# B&R Automation Studio project Parker_BMM_ST_V5_3147_V12 (part 31)

#### modem.c
```c
/********************************************************************
 * COPYRIGHT --  B&R China
 ********************************************************************
 * Program: modem
 * File: modem.c
 * Author: lijianjun
 * Created: March 06, 2013
 ********************************************************************
 * Implementation of program modem --- modem remote communication  control
 ********************************************************************/

#ifdef _DEFAULT_INCLUDES
	#include <AsDefault.h>
#endif

#include <bur/plctypes.h>
#include <string.h>
#include "edge.h"

/**************************************************************************************
** 					 	     define 								                 **
**************************************************************************************/
#define	BRTRSM_COMMAND_CHAR_MAXCOUT			20
#define	BRTRSM_COMMAND_MAXCOUT					20

#define  BRTRSM_EXCHANGEDATA_CHAR_MAXCOUT		64

#define  BRTRSM_ERR_FUB_BUSY		0xFFFF

/**************************************************************************************
** 					 	     function 								                 **
**************************************************************************************/
UINT	BRFindString(char * p,char * str);

/**************************************************************************************
**     	        		I N I T U P  O F   T H E   T A S K 		 				     **
**************************************************************************************/
 _INIT void init ( void )
 {
	 BRInitStep		= 1000;
	 BRStep			= 0;
 }

 /**************************************************************************************
**        				C Y C L I C   P A R T   O F   T H E   T A S K  				 **
**************************************************************************************/

 _CYCLIC void cyclic ( void )
 {

	switch	(BRInitStep)
	{
		case 1000:

			cmdModem		=0;

			strcpy(FmDevice,"IF1");
			#ifdef __i386__

			strcpy(FmMode,"/PHY=RS232 /BD=57600 /PA=N /DB=8 /SB=1");

			#else

			strcpy(FmMode,"57600,N,8,1,RS232");

			#endif

			i	=0;

			strcpy(AcT[i++].Command,"AT&F");	  /* DEFAULT SETTING  */
			strcpy(AcT[i++].Command,"ATS0=1");
			strcpy(AcT[i++].Command,"ATS37=9");
			strcpy(AcT[i++].Command,"AT&C0");
			strcpy(AcT[i++].Command,"AT&D0");
			strcpy(AcT[i++].Command,"AT&K0");
			strcpy(AcT[i++].Command,"AT&Q0");
			strcpy(AcT[i++].Command,"AT&W0");
			strcpy(AcT[i++].Command,"AT&Y0");

			ATCommandCount = i;

			BRInitStep	   = 2000;

			break;
		case 2000:
			if (0 == BRStep && 1 == cmdModem)
			{
				gMachineInfo.Modem_Ok	= 0;
				BRStep		= 1000;
				BRInitStep	= 3000;
			}
			break;
		case 3000:
			Status	=BRFindString(BRReadBuf,BRWriteBuf);
			break;
		default:
         break;
	}
	switch	(BRStep)
	{
		case 1000:

			BRFRMxopen.device	= (unsigned long)&FmDevice;
			BRFRMxopen.mode		= (unsigned long)&FmMode;
			BRFRMxopen.enable	= 1;

			FRM_xopen(&BRFRMxopen);

			if(0 == BRFRMxopen.status)
			{
				BRStep	= 2000;
			}

			break;

		case 2000:

			BRFRMctrl.enable	= 1;
			BRFRMctrl.ident		= BRFRMxopen.ident;
			BRFRMctrl.ioctrl	= 0x12;
			BRFRMctrl.inarg		= 1;

			FRM_ctrl(&BRFRMctrl);

			BRFRMctrl.enable	= 1;
			BRFRMctrl.ident		= BRFRMxopen.ident;
			BRFRMctrl.ioctrl	= 0x27;

			FRM_ctrl(&BRFRMctrl);

			BRStep	= 3000;

			break;
		case 3000:

			memset(BRWriteBuf,0,BRTRSM_EXCHANGEDATA_CHAR_MAXCOUT);
			strcpy(BRWriteBuf,"AT&F");
			BRWriteBuf[4]	= 0x0D;
			BRWriteBuf[5]	= 0x00;

			BRFRMwrite.enable	= 1;
			BRFRMwrite.ident	= BRFRMxopen.ident;
			BRFRMwrite.buffer	= (unsigned long)BRWriteBuf;
			BRFRMwrite.buflng	= strlen(BRWriteBuf);

			FRM_write(&BRFRMwrite);

			if(0 == BRFRMwrite.status)
			{
				BRStep = 3200;
			}

			break;
		case 3200:
			memset(BRWriteBuf,0,BRTRSM_EXCHANGEDATA_CHAR_MAXCOUT);
			strcpy(BRWriteBuf,"ATE0");
			BRWriteBuf[4]	= 0x0D;
			BRWriteBuf[5]	= 0x00;

			BRFRMwrite.enable	= 1;
			BRFRMwrite.ident	= BRFRMxopen.ident;
			BRFRMwrite.buffer	= (unsigned long)BRWriteBuf;
			BRFRMwrite.buflng	= strlen(BRWriteBuf);

			FRM_write(&BRFRMwrite);

			if(0 == BRFRMwrite.status)
			{
				BRStep = 3600;
			}

			break;
		case 3600:
			memset(BRWriteBuf,0,BRTRSM_EXCHANGEDATA_CHAR_MAXCOUT);
			strcpy(BRWriteBuf,"AT&Q0");
			BRWriteBuf[4]	= 0x0D;
			BRWriteBuf[5]	= 0x00;

			BRFRMwrite.enable	= 1;
			BRFRMwrite.ident	= BRFRMxopen.ident;
			BRFRMwrite.buffer	= (unsigned long)BRWriteBuf;
			BRFRMwrite.buflng	= strlen(BRWriteBuf);

			FRM_write(&BRFRMwrite);

			if(0 == BRFRMwrite.status)
			{
				BRStep = 4000;
			}
			break;
		case 4000:

			BRFRMread.enable = 1;
			BRFRMread.ident	 = BRFRMxopen.ident;

			FRM_read(&BRFRMread);

			if(0 == BRFRMread.status)
			{
				if(BRFRMread.buflng<=BRTRSM_EXCHANGEDATA_CHAR_MAXCOUT)
				{
					memcpy(BRReadBuf,(void*)BRFRMread.buffer,BRFRMread.buflng);		/* copy received data */

					BRFRMrbuf.enable	= 1;
					BRFRMrbuf.ident		= BRFRMxopen.ident;
					BRFRMrbuf.buffer	= BRFRMread.buffer;
					BRFRMrbuf.buflng	= BRFRMread.buflng;

					FRM_rbuf(&BRFRMrbuf);											/* release buffer again */

					if(BRFindString(BRReadBuf,"OK")==1)
					{
						CurrentAT	= 0;
						BRStep		= 5000;
					}
					else
					{
						BRStep		= 3000;
					}
				}
			}

			break;
		case 5000:

			memset(BRWriteBuf,0,BRTRSM_EXCHANGEDATA_CHAR_MAXCOUT);
			strcpy(BRWriteBuf,AcT[CurrentAT].Command);
			TempLength	=strlen(BRWriteBuf);
			BRWriteBuf[TempLength]		= 0x0D;
			BRWriteBuf[TempLength+1]	= 0x00;

			TempLength++;

			BRFRMwrite.enable		=1;
			BRFRMwrite.ident		=BRFRMxopen.ident;
			BRFRMwrite.buffer		=(unsigned long)BRWriteBuf;
			BRFRMwrite.buflng		=strlen(BRWriteBuf);

			FRM_write(&BRFRMwrite);

			if(BRFRMwrite.status==0)
			{
				BRStep			=6000;
			}

			break;
		case 6000:

			BRFRMread.enable		=1;
			BRFRMread.ident			=BRFRMxopen.ident;

			FRM_read(&BRFRMread);

			if(BRFRMread.status==0)
			{
				if(BRFRMread.buflng<=BRTRSM_EXCHANGEDATA_CHAR_MAXCOUT)
				{
					memcpy(BRReadBuf,(void*)BRFRMread.buffer,BRFRMread.buflng);		/* copy received data */

					BRFRMrbuf.enable	=1;
					BRFRMrbuf.ident		=BRFRMxopen.ident;
					BRFRMrbuf.buffer	=BRFRMread.buffer;
					BRFRMrbuf.buflng	=BRFRMread.buflng;

					FRM_rbuf(&BRFRMrbuf);											/* release buffer again */

					if(BRFindString(BRReadBuf,"OK")==1)
					{
						CurrentAT++;
						if(CurrentAT>=ATCommandCount)
						{
							BRStep		=7000;
							break;
						}
					}
					BRStep			=5000;

				}
			}
			break;
		case 7000:

			BRFRMclose.enable	=1;
			BRFRMclose.ident	=BRFRMxopen.ident;

			FRM_close(&BRFRMclose);

			BRStep	= 8000;

			break;

		case 8000:
			cmdModem		=0;
			gMachineInfo.Modem_Ok =1;
			BRStep		    =0;

			break;
		default:
         break;
	}

 }
/**************************************************************************************
** 					 	     function 								                 **
**************************************************************************************/
UINT	BRFindString(char * p,char * str)
{
   UINT pLength,strLength,i,j;

   pLength	   =strlen(p);
   strLength	=strlen(str);

   if(strLength==0)
      return 0;
   if(pLength==0)
      return 0;

   j		=0;

   for(i=0;i<pLength;i++)
   {
      if(p[i]==str[j])
      {
         j++;
         if(j>=strLength)
         {
            return 1;
         }
      }
      else
      {
         j		=0;
         if(p[i]==str[j])
         {
            j++;
            if(j>=strLength)
            {
               return 1;
            }
         }
      }
   }

   return 0;
}
```

#### modem.var
```iecst
VAR
	cmdModem : BOOL;
	BRInitStep : UINT;
	BRStep : UINT;
	Status : UINT;
	i : UINT;
	ATCommandCount : UINT;
	CurrentAT : UINT;
	TempLength : UINT;
	BRReadBuf : STRING[80];
	BRWriteBuf : STRING[80];
	FmDevice : STRING[80];
	FmMode : STRING[80];
	BRFRMwrite : FRM_write;
	BRFRMread : FRM_read;
	BRFRMctrl : FRM_ctrl;
	BRFRMxopen : FRM_xopen;
	BRFRMrbuf : FRM_rbuf;
	BRFRMclose : FRM_close;
	AcT : ARRAY[0..19] OF BRTransfer;
END_VAR
```

### Program Logical/comm/mbusMaster (ANSIC, version 1.00.0) - communication with frequency inventor

#### mbusMaster.c - Implementation code
```c
/********************************************************************
 * COPYRIGHT --
 ********************************************************************
 * Program: mbusMaster
 * File: mbusMaster.c
 * Author: lij
 * Created: December 12, 2014
 ********************************************************************
 * Implementation of program mbusMaster
 ********************************************************************/

#include <bur/plctypes.h>
#include <string.h>

#ifdef _DEFAULT_INCLUDES
	#include <AsDefault.h>
#endif

#define	_AR_I386_AUTOMATION_STUDIO_   1

void _INIT mbusMasterINIT(void)
{
	/* TODO: Add code here */

   ascii = 0;    /* 0 = RTU / 1 = ASCII */

#ifdef _AR_I386_AUTOMATION_STUDIO_
   strcpy(sDeviceName, "SL1.SS1.IF1.ST2.IF1");
   if (!ascii)
   {
      strcpy(sModeName, "PHY=RS485 /BD=19200 /PA=O /DB=8");
   }
   else
   {
      strcpy(sModeName, "PHY=RS485 /BD=19200 /PA=O /DB=7");
   }
#else
   strcpy(sDeviceName, "SS1.IF1");
   if (!ascii)
   {
      strcpy(sModeName, "RS232,19200,E,8,1");
   }
   else
   {
      strcpy(sModeName, "RS232,19200,E,8,1");
   }
#endif

   strcpy(sConfigName, "mb_cmd");

   timeout  = 500; /* 500ms */

   /* modbus - Slave open */
   MOpen.enable   = 1;
   MOpen.pDevice  = (UDINT) &sDeviceName[0];
   MOpen.pMode    = (UDINT) &sModeName[0];
   MOpen.pConfig  = (UDINT) &sConfigName[0];
   MOpen.timeout  = timeout;
   MOpen.ascii = ascii;

   MBMOpen(&MOpen);

   statusMOpen = MOpen.status;
   if (!statusMOpen)
   {
      ident    = MOpen.ident;
      fMOpen   = 0;
      fMaster  = 1;
      fMClose  = 0;
   }
   else
   {
      fMaster = 0;
      ident   = 0;
      fMOpen  = 1;
   }

   fMClose = 0;
}

void _CYCLIC mbusMasterCYCLIC(void)
{
	/* TODO: Add code here */

   if(fMOpen)
   {
      /* modbus - Master open */
      MOpen.enable   = 1;
      MOpen.pDevice  = (UDINT) &sDeviceName[0];
      MOpen.pMode    = (UDINT) &sModeName[0];
      MOpen.pConfig  = (UDINT) &sConfigName[0];
      MOpen.timeout  = timeout;
      MOpen.ascii    = ascii;

      MBMOpen(&MOpen);

      statusMOpen = MOpen.status;
      if (!statusMOpen)
      {
         ident   = MOpen.ident;
         fMOpen  = 0;
         fMaster = 1;
         fMClose = 0;
      }
      else
      {
         fMaster = 0;
         ident   = 0;
         fMOpen  = 1;
      }
   }

   if(fMaster)
   {
      /* modbus - Master */
      Master.enable = 1;
      Master.ident  = ident;
      MBMaster(&Master);

      statusMaster= Master.status;
      execute     = Master.execute;
      recordnum   = Master.recordnum;

      if (!statusMaster)
      {
         fMaster = 1;
      }
   }

   if(fMClose)
   {
      fMaster = 0;
      fMClose = 0;

      /* modbus - Master close */
      MClose.enable = 1;
      MClose.ident  = ident;
      MBMClose(&MClose);

      statusMClose = MClose.status;
      if (!statusMClose)
      {
         ident  = 0;
         fMOpen = 0;
      }
   }
}

void _EXIT mbusMasterEXIT(void)
{
	/* TODO: Add code here */

   MClose.enable   = 1;
   MClose.ident    = ident;
   MBMClose(&MClose);
}
```

#### mbusMaster.var - Local variables
```iecst
(********************************************************************
 * COPYRIGHT --
 ********************************************************************
 * Program: mbusMaster
 * File: mbusMaster.var
 * Author: lij
 * Created: December 12, 2014
 ********************************************************************
 * Local variables of program mbusMaster
 ********************************************************************)
VAR
	MOpen : MBMOpen;
	Master : MBMaster;
	MClose : MBMClose;
	fMOpen : BOOL;
	fMaster : BOOL;
	fMClose : BOOL;
	ascii : USINT;
	statusMOpen : UINT;
	statusMaster : UINT;
	statusMClose : UINT;
	timeout : UINT;
	ident : UDINT;
	execute : UDINT;
	recordnum : UDINT;
	sDeviceName : STRING[80];
	sModeName : STRING[80];
	sConfigName : STRING[80];
END_VAR
```

### Data object Logical/comm/mb_cmd (Simple) - A simple data object.

#### mb_cmd.dat
```
(********************************************************************
 * COPYRIGHT --
 ********************************************************************
 * Data object: mb_cmd
 * File: mb_cmd.dat
 * Author: lij
 * Created: December 12, 2014
 ********************************************************************
 * Data object file: mb_cmd.dat
 ********************************************************************)
; ---------------------------------------------------------------------------
; SanKen VM06 系列选件板
; MODBUS-RTU
; MODBUS command table
; ---------------------------------------------------------------------------
; Modbus Function Code description
; ---------------------------------------------------------------------------
; 功能编码	名称
; 0x03	    读控制继电器
; 0x04	    读输入继电器
; 0x06	    写信号继电器
; 0x10	    Preset Multiple Register
; ---------------------------------------------------------------------------
; ---------------------------------------------------------------------------

; ---------------------------------------------------------------------------
; ---------------------------------------------------------------------------
;         1         2         3                        1         2         3
;1234567890123456789012345678901              1234567890123456789012345678901
;"                               ", 03, $02, "LocalPV3                       ", 0000, 0800    ;read from MB4[x], block read supported
;"                               ", 06, $02, "LocalPV6[0]                    ", 0000, 0001    ;function code 6:write to MB4[x]
;"                               ", 16, $02, "LocalPV16                      ", 0000, 0200    ;EventPV16
;|                                 |    |    |                                  |     |
;|                                 |    |    |                                  |     |
;Event variable                    |    |    Variable name on this station      |     Data Length to be read or written[WORD]
;                                  |    Node number [BYTE](server?)             Modbus offset
;                                  Modbus function code [BYTE]                  on slave station [WORD]
; ---------------------------------------------------------------------------
; ---------------------------------------------------------------------------

;1234567890123456789012345678901             1234567890123456789012345678901

;Slave 1:	Main   Extruder		SanKen VM06-0150-N4
"                               ", 06, $01, "gMbusCom[0].WriteFrequency      ", 1000, 0001
"                               ", 06, $01, "gMbusCom[0].WriteCommand        ", 1001, 0001
"                               ", 06, $01, "gMbusCom[0].WriteAckAlarm       ", 1002, 0001
"                               ", 03, $01, "gMbusCom[0].ReadCurrent         ", 2003, 0001
"                               ", 03, $01, "gMbusCom[0].ReadFrequency       ", 2002, 0001
"                               ", 03, $01, "gMbusCom[0].ReadVoltage         ", 2014, 0001
"                               ", 03, $01, "gMbusCom[0].ReadAlarmNum        ", 2000, 0001
"                               ", 03, $01, "gMbusCom[0].ReadStatus          ", 2008, 0002
; ---------------------------------------------------------------------------
; ---------------------------------------------------------------------------
;Slave 2:	AUX1   Extruder		SanKen VM06-0150-N4
"                               ", 06, $02, "gMbusCom[1].WriteFrequency      ", 1000, 0001
"                               ", 06, $02, "gMbusCom[1].WriteCommand        ", 1001, 0001
"                               ", 06, $02, "gMbusCom[1].WriteAckAlarm       ", 1002, 0001
"                               ", 03, $02, "gMbusCom[1].ReadCurrent         ", 2003, 0001
"                               ", 03, $02, "gMbusCom[1].ReadFrequency       ", 2002, 0001
"                               ", 03, $02, "gMbusCom[1].ReadVoltage         ", 2014, 0001
"                               ", 03, $02, "gMbusCom[1].ReadAlarmNum        ", 2000, 0001
"                               ", 03, $02, "gMbusCom[1].ReadStatus          ", 2008, 0002
; ---------------------------------------------------------------------------
; ---------------------------------------------------------------------------
```

### Program Logical/comm/epl (ANSIC)

#### epl.c - Init, cyclic, exit code
```c
#include <bur/plctypes.h>

#ifdef _DEFAULT_INCLUDES
	#include <AsDefault.h>
#endif

void _INIT eplInit(void)
{
	EPLInverter[0].cmd.readNode = 1;
	EPLInverter[1].cmd.readNode = 1;
	EPLInverter[2].cmd.readNode = 1;
	EPLInverter[3].cmd.readNode = 1;

	strcpy(&sDevice[0],"SL1.IF1");
	strcpy(&sDevice[1],"SL1.IF1");
	strcpy(&sDevice[2],"SL1.IF1");
	strcpy(&sDevice[3],"SL1.IF1");

	strcpy(&sDeviceAExtr,"SL1.IF1");

	uIndexOffset = 7;

	/*Albert*/

	uCountTimerA = 100;/*1 second*/
	uCountTimerB = 100;/*1 second*/
	uCountTimerC = 100;/*1 second*/
	uCountTimerV = 100;/*1 second*/

	uIndexA = 0;
	uIndexB = 0;
	uIndexC = 0;
	uIndexV = 0;
}

void _CYCLIC eplCyclic(void)
{
//	int i;
//	for(i=0;i<4;i++)/*For extruder A , B , C and V*/
//	{
//		if(EPLInverter[i].para.nodeNr != 0)
//		{
//			if(EPLInverter[i].state = EPL_WAIT)
//			{
//				EPLInverter[i].cmd.bReadObj = 1;/*read command*/
//				if (0 == uIndexRead[i])
//				{
//					EPLInverter[i].para.MotorPower = (INT) EPLInverter[i].para.readData;
//					uIndexRead[i] = uIndexRead[i]+10;
//					EPLInverter[i].cmd.index = 0x2002;
//					EPLInverter[i].cmd.subindex = 0x9;
//				}
//				else if (10 == EPLInverter[i].cmd.index)
//				{
//					EPLInverter[i].para.MotorVoltage = (INT) EPLInverter[i].para.readData;
//					uIndexRead[i] = 0;
//					EPLInverter[i].cmd.index = 0x2002;
//					EPLInverter[i].cmd.subindex = 0xC;
//				}
//			}
//		}
//		switch (EPLInverter[i].state)
//		{
//			case EPL_WAIT: /*state to wait for user Commands*/
//
//				if(1 == EPLInverter[i].cmd.readNode)
//				{
//					EPLInverter[i].cmd.readNode = 0;
//					EPLInverter[i].state = EPL_READ_NODE;
//				}
//				else if(1 == EPLInverter[i].cmd.bReadObj)
//				{
//					EPLInverter[i].cmd.readThresholdCnt = 0;
//					EPLInverter[i].state = EPL_READ_OE;
//				}
//				else if(1 == EPLInverter[i].cmd.bWriteObj)
//				{
//					EPLInverter[i].cmd.bWriteObj = 0;
//					EPLInverter[i].state = EPL_WRITE_OE;
//				}
//
//				break;
//			case EPL_READ_NODE:/*state to read the local Powerlink node number*/
//				EPLInverter[i].fub.fnEplGetLocalNodeID.enable = 1;
//				EPLInverter[i].fub.fnEplGetLocalNodeID.pDevice = (UDINT) &sDevice[i];
//
//				if(EPLInverter[i].fub.fnEplGetLocalNodeID.status == 0)
//				{
//					EPLInverter[i].para.nodeNr = EPLInverter[i].fub.fnEplGetLocalNodeID.nodeid;
//					EPLInverter[i].fub.fnEplGetLocalNodeID.enable = 0;
//					EPLInverter[i].state = EPL_WAIT;
//				}
//				else if(EPLInverter[i].fub.fnEplGetLocalNodeID.status == ERR_FUB_BUSY)
//				{
//					EPLInverter[i].state = EPL_READ_NODE;/*creating not finished --> do again*/
//				}
//				else if (EPLInverter[i].fub.fnEplGetLocalNodeID.status == ERR_FUB_ENABLE_FALSE)
//				{
//					/*FUB is disabled*/
//				}
//				else
//				{
//					EPLInverter[i].state = EPL_ERROR;
//				}
//
//
//				break;
//			case EPL_READ_OE:/*state to read an object entry*/
//
//				EPLInverter[i].fub.fnEplSDORead.enable = 1;
//				EPLInverter[i].fub.fnEplSDORead.pDevice = (UDINT) &sDevice[i];
//				EPLInverter[i].fub.fnEplSDORead.node = uIndexOffset + i;
//				EPLInverter[i].fub.fnEplSDORead.index = EPLInverter[i].cmd.index;
//				EPLInverter[i].fub.fnEplSDORead.subindex = EPLInverter[i].cmd.subindex;
//				EPLInverter[i].fub.fnEplSDORead.pData = (UDINT) &EPLInverter[i].para.readData;
//				EPLInverter[i].fub.fnEplSDORead.datalen = sizeof(EPLInverter[i].para.readData);
//
//				if(EPLInverter[i].fub.fnEplSDORead.status == 0)
//				{
//					EPLInverter[i].fub.fnEplSDORead.enable = 0;
//					EPLInverter[i].state = EPL_WAIT;
//				}
//				else if(EPLInverter[i].fub.fnEplSDORead.status == ERR_FUB_BUSY)
//				{
//					EPLInverter[i].state = EPL_READ_OE;
//				}
//				else if(EPLInverter[i].fub.fnEplSDORead.status == ERR_FUB_ENABLE_FALSE)
//				{
//				}
//				else
//				{
//					EPLInverter[i].state = EPL_ERROR;
//				}
//
//				break;
//			case EPL_WRITE_OE:/*state to write an object entry*/
//				break;
//			case EPL_ERROR:/*State when an error occured*/
//				break;
//		}
//	}

//	if(bTestRead)
//	{
		for(i=0;i<4;i++)
		{
			if(EPLInverter[i].para.nodeNr != 0)
			{
				if(EPLInverter[i].state == EPL_WAIT)
				{
					EPLInverter[i].cmd.bReadObj = 1;/*read command*/
					if (0 == uIndexRead[i])
					{
						EPLInverter[i].para.EnergyCons = (INT) EPLInverter[i].para.readData;
//						EPLInverter[i].para.MotorPower = (INT) EPLInverter[i].para.readData;
						uIndexRead[i] = uIndexRead[i]+10;
						EPLInverter[i].cmd.index = 0x2002;
						EPLInverter[i].cmd.subindex = 0x9;
					}
					else if (10 == uIndexRead[i])
					{
						EPLInverter[i].para.MotorVoltage = (INT) EPLInverter[i].para.readData;
//						EPLInverter[i].para.MotorVoltage = (INT) EPLInverter[i].para.readData;
						uIndexRead[i] = uIndexRead[i]+10;
						EPLInverter[i].cmd.index = 0x2002;
						EPLInverter[i].cmd.subindex = 0xC;
					}
					else if(20 == uIndexRead[i])
					{
						EPLInverter[i].para.MotorPower = (INT) EPLInverter[i].para.readData;
//						EPLInverter[i].para.EnergyCons = (INT) EPLInverter[i].para.readData;
						uIndexRead[i] = 0;
						EPLInverter[i].cmd.index = 0x2002;
						EPLInverter[i].cmd.subindex = 0x1F;
					}
				}
			}
			switch (EPLInverter[i].state)
			{
				case EPL_WAIT: /*state to wait for user Commands*/

					if(1 == EPLInverter[i].cmd.readNode)
					{
						EPLInverter[i].cmd.readNode = 0;
						EPLInverter[i].state = EPL_READ_NODE;
					}
					else if(1 == EPLInverter[i].cmd.bReadObj)
					{
						EPLInverter[i].cmd.bReadObj = 0;
						EPLInverter[i].state = EPL_READ_OE;
					}
					else if(1 == EPLInverter[i].cmd.bWriteObj)
					{
						EPLInverter[i].cmd.bWriteObj = 0;
						EPLInverter[i].state = EPL_WRITE_OE;
					}

					break;
				case EPL_READ_NODE:/*state to read the local Powerlink node number*/
					EPLInverter[i].fub.fnEplGetLocalNodeID.enable = 1;
					EPLInverter[i].fub.fnEplGetLocalNodeID.pDevice = (UDINT) &sDevice[i];

					if(EPLInverter[i].fub.fnEplGetLocalNodeID.status == 0)
					{
						EPLInverter[i].para.nodeNr = EPLInverter[i].fub.fnEplGetLocalNodeID.nodeid;
						EPLInverter[i].fub.fnEplGetLocalNodeID.enable = 0;
						EPLInverter[i].state = EPL_WAIT;

					}
					else if(EPLInverter[i].fub.fnEplGetLocalNodeID.status == ERR_FUB_BUSY)
					{
						EPLInverter[i].state = EPL_READ_NODE;/*creating not finished --> do again*/
					}
					else if (EPLInverter[i].fub.fnEplGetLocalNodeID.status == ERR_FUB_ENABLE_FALSE)
					{
						/*FUB is disabled*/
					}
					else
					{
						EPLInverter[i].state = EPL_ERROR;
					}

					break;
				case EPL_READ_OE:/*state to read an object entry*/

					EPLInverter[i].fub.fnEplSDORead.enable = 1;
					EPLInverter[i].fub.fnEplSDORead.pDevice = (UDINT) &sDeviceAExtr;
					EPLInverter[i].fub.fnEplSDORead.node = uIndexOffset;
					EPLInverter[i].fub.fnEplSDORead.index = EPLInverter[i].cmd.index;
					EPLInverter[i].fub.fnEplSDORead.subindex = EPLInverter[i].cmd.subindex;
					EPLInverter[i].fub.fnEplSDORead.pData = (UDINT) &EPLInverter[i].para.readData;
					EPLInverter[i].fub.fnEplSDORead.datalen = sizeof(EPLInverter[i].para.readData);

					if(EPLInverter[i].fub.fnEplSDORead.status == 0)
					{
						EPLInverter[i].fub.fnEplSDORead.enable = 0;
						EPLInverter[i].state = EPL_WAIT;
					}
					else if(EPLInverter[i].fub.fnEplSDORead.status == ERR_FUB_BUSY)
					{
						EPLInverter[i].state = EPL_READ_OE;
					}
					else if(EPLInverter[i].fub.fnEplSDORead.status == ERR_FUB_ENABLE_FALSE)
					{
					}
					else
					{
						EPLInverter[i].state = EPL_ERROR;
					}

					break;
				case EPL_WRITE_OE:/*state to write an object entry*/
					break;
				case EPL_ERROR:/*State when an error occured*/
					break;
			}
		}
//	}
//	else
//	{
//		EPLInverter[i].fub.fnEplSDORead.enable = 0;
//		EPLInverter[i].fub.fnEplGetLocalNodeID.enable = 0;
//		EPLInverter[i].fub.fnEplSDOWrite.enable = 0;
//	}

	/*P84 Inverter power consumption*/

	/*Albert Add power consumption function*/

	/*----A Extruder-----*/
	switch (uStepPowerA)
	{
		case 0:/*Weit step*/
		if(gMachineInfo.Auto)
//			if(bTestAuto)
			{
				fnTON_10msA.IN = 1;
				fnTON_10msA.PT = uCountTimerA;
				uStepPowerA = 10;
			}
			break;
		case 10:/*Start Timer*/
			if(fnTON_10msA.Q)
			{
				fnTON_10msA.IN = 0;
				uIndexA++;
				uStepPowerA = 20;
			}
			if(0 == gMachineInfo.Auto)
//			if(0 == bTestAuto)
			{
				uIndexA	=	0;
				fnTON_10msA.IN = 0;
				uStepPowerA = 0;
			}
			break;
		case 20:/*Get value*/
			if(uIndexA > 59)
			{
				uIndexA = 0;
				rPowerTotalA += (rPowerTotalPerSecA/3600);
			}
			rPowerTotalPerSecA = 0;

			rActCurrentA[uIndexA] = gExtruderACtrl.InverterStatus.Current/10;/*Change unit from 0.1A to 1A*/
			rActVoltageA[uIndexA] = EPLInverter[0].para.MotorVoltage;
	//		rActCurrentA[uIndexA] = mcParID_Value.readPar.actCurrent;
	//		rActVoltageA[uIndexA] = mcParID_Value.readPar.actUDC;
	//		rActCurrentA[uIndexA] = rTestCurrent;
	//		rActVoltageA[uIndexA] = rTestVoltage;

			uStepPowerA = 30;

			break;
		case 30:/*Calculate*/
			rPowerA[uIndexA] = (rActCurrentA[uIndexA] * rActVoltageA[uIndexA])/1000;
			for(i_A=0;i_A<60;i_A++)
			{
				rPowerTotalPerSecA += rPowerA[i_A];
			}
			rPowerPerMinA= rPowerTotalPerSecA/60;
			uStepPowerA = 0;
			break;
	}

	/*Function call*/
	TON_10ms(&fnTON_10msA);

	/*Reset Function*/
	if(bCleanPowerA)
	{
		iClickTimeA--;
		if(iClickTimeA <= 0)
		{
			bCleanPowerA = 0;
			rPowerTotalA = 0;
			rPowerPerMinA = 0;
		}
	}
	else
	{
		iClickTimeA = 10;
	}

	/*----B Extruder-----*/
	switch (uStepPowerB)
	{
		case 0:/*Weit step*/
			if(gMachineInfo.Auto)
			{
				fnTON_10msB.IN = 1;
				fnTON_10msB.PT = uCountTimerB;
				uStepPowerB = 10;
			}
			break;
		case 10:/*Start Timer*/
			if(fnTON_10msB.Q)
			{
				fnTON_10msB.IN = 0;
				uIndexB++;
				uStepPowerB = 20;
			}
			if(0 == gMachineInfo.Auto)
			{
				uIndexB	=	0;
				fnTON_10msB.IN = 0;
				uStepPowerB = 0;
			}
			break;
		case 20:/*Get value*/
			if(uIndexB > 59)
			{
				uIndexB = 0;
				rPowerTotalB += (rPowerTotalPerSecB/3600);
			}
			rPowerTotalPerSecB = 0;

			rActCurrentB[uIndexB] = gExtruderBCtrl.InverterStatus.Current/10;/*Change unit from 0.1A to 1A*/
			rActVoltageB[uIndexB] = EPLInverter[1].para.MotorVoltage;
			//		rActCurrentA[uIndexA] = mcParID_Value.readPar.actCurrent;
			//		rActVoltageA[uIndexA] = mcParID_Value.readPar.actUDC;

			uStepPowerB = 30;

			break;
		case 30:/*Calculate*/
			rPowerB[uIndexB] = (rActCurrentB[uIndexB] * rActVoltageB[uIndexB])/1000;
			for(i_B=0;i_B<60;i_B++)
			{
				rPowerTotalPerSecB += rPowerB[i_B];
			}
			rPowerPerMinB = rPowerTotalPerSecB/60;
			uStepPowerB = 0;
			break;
	}
	/*Calculate total power*/
//	switch (uStepPowerHourB)
//	{
//		case 0:
//			if(gMachineInfo.Auto)
//			{
//				fnTON_10msB_HR.IN = 1;
//				fnTON_10msB_HR.PT = 60000;
//				uStepPowerHourB = 10;
//			}
//			break;
//		case 10:
//			if(fnTON_10msB_HR.Q)
//			{
//				fnTON_10msB_HR.IN = 0;
//				uStepPowerHourB = 20;
//			}
//			if(0 == gMachineInfo.Auto)
//			{
//				fnTON_10msB_HR.IN = 1;
//				fnTON_10msB_HR.PT = 60000;
//				uStepPowerHourB = 10;
//			}
//			break;
//		case 20:
//			rPowerTotalB = rPowerTotalB + (rPowerPerSecB/6);
//			uStepPowerHourB = 30;
//			break;
//		case 30:
//			uStepPowerHourB = 0;
//			break;
//	}

	/*Function call*/
	TON_10ms(&fnTON_10msB);
	TON_10ms(&fnTON_10msB_HR);

	/*Reset Function*/
	if(bCleanPowerB)
	{
		iClickTimeB--;
		if(iClickTimeB <= 0)
		{
			bCleanPowerB = 0;
			rPowerTotalB = 0;
			rPowerPerMinB = 0;
		}
	}
	else
	{
		iClickTimeB = 10;
	}

	/*----C Extruder-----*/
	switch (uStepPowerC)
	{
		case 0:/*Weit step*/
			if(gMachineInfo.Auto)
			{
				fnTON_10msC.IN = 1;
				fnTON_10msC.PT = uCountTimerC;
				uStepPowerC = 10;
			}
			break;
		case 10:/*Start Timer*/
			if(fnTON_10msC.Q)
			{
				fnTON_10msC.IN = 0;
				uIndexC++;
				uStepPowerC = 20;
			}
			if(0 == gMachineInfo.Auto)
			{
				uIndexC	=	0;
				fnTON_10msC.IN = 0;
				uStepPowerC = 0;
			}
			break;
		case 20:/*Get value*/
			if(uIndexC > 59)
			{
				uIndexC = 0;
				rPowerTotalC += rPowerTotalPerSecC;
//				rPowerPerHrC = rPowerPerSecC * 60 * 60;
			}
			rPowerTotalPerSecC = 0;

			rActCurrentC[uIndexC] = gExtruderCCtrl.InverterStatus.Current/10;/*Change unit from 0.1A to 1A*/
			rActVoltageC[uIndexC] = EPLInverter[2].para.MotorVoltage;
			//		rActCurrentA[uIndexA] = mcParID_Value.readPar.actCurrent;
			//		rActVoltageA[uIndexA] = mcParID_Value.readPar.actUDC;

			uStepPowerC = 30;

			break;
		case 30:/*Calculate*/
			rPowerC[uIndexC] = (rActCurrentC[uIndexC] * rActVoltageC[uIndexC])/1000;
			for(i_C=0;i_C<60;i_C++)
			{
				rPowerTotalPerSecC += rPowerC[i_C];
			}
			rPowerPerMinC = rPowerTotalPerSecC/60;
			uStepPowerC = 0;
			break;
	}

	/*Function call*/
	TON_10ms(&fnTON_10msC);

	/*Reset Function*/
	if(bCleanPowerC)
	{
		iClickTimeC--;
		if(iClickTimeC <= 0)
		{
			bCleanPowerC = 0;
			rPowerTotalC = 0;
			rPowerPerMinC = 0;
		}
	}
	else
	{
		iClickTimeC = 10;
	}

	/*----V Extruder-----*/
	switch (uStepPowerV)
	{
		case 0:/*Weit step*/
			if(gMachineInfo.Auto)
			{
				fnTON_10msV.IN = 1;
				fnTON_10msV.PT = uCountTimerV;
				uStepPowerV = 10;
			}
			break;
		case 10:/*Start Timer*/
			if(fnTON_10msV.Q)
			{
				fnTON_10msV.IN = 0;
				uIndexV++;
				uStepPowerV = 20;
			}
			if(0 == gMachineInfo.Auto)
			{
				uIndexV	=	0;
				fnTON_10msV.IN = 0;
				uStepPowerV = 0;
			}
			break;
		case 20:/*Get value*/
			if(uIndexV > 59)
			{
				uIndexV = 0;
				rPowerTotalV += (rPowerTotalPerSecV/3600);
			}
			rPowerTotalPerSecV = 0;

			rActCurrentV[uIndexV] = gExtruderVCtrl.InverterStatus.Current/10;/*Change unit from 0.1A to 1A*/
			rActVoltageV[uIndexV] = EPLInverter[3].para.MotorVoltage;
			//		rActCurrentA[uIndexA] = mcParID_Value.readPar.actCurrent;
			//		rActVoltageA[uIndexA] = mcParID_Value.readPar.actUDC;

			uStepPowerV = 30;

			break;
		case 30:/*Calculate*/
			rPowerV[uIndexV] = (rActCurrentV[uIndexV] * rActVoltageV[uIndexV])/1000;
			for(i_V=0;i_V<60;i_V++)
			{
				rPowerTotalPerSecV += rPowerV[i_V];
			}
			rPowerPerMinV = rPowerTotalPerSecV/60;
			uStepPowerV = 0;
			break;
	}

	/*Function call*/
	TON_10ms(&fnTON_10msV);

	/*Reset Function*/
	if(bCleanPowerV)
	{
		iClickTimeV--;
		if(iClickTimeV <= 0)
		{
			bCleanPowerV = 0;
			rPowerTotalV = 0;
			rPowerPerMinV = 0;
		}
	}
	else
	{
		iClickTimeV = 10;
	}

	/*Function Call*/

	EplGetLocalNodeID(&EPLInverter[0].fub.fnEplGetLocalNodeID);
	EplGetLocalNodeID(&EPLInverter[1].fub.fnEplGetLocalNodeID);
	EplGetLocalNodeID(&EPLInverter[2].fub.fnEplGetLocalNodeID);
	EplGetLocalNodeID(&EPLInverter[3].fub.fnEplGetLocalNodeID);

	EplSDORead(&EPLInverter[0].fub.fnEplSDORead);
	EplSDORead(&EPLInverter[1].fub.fnEplSDORead);
	EplSDORead(&EPLInverter[2].fub.fnEplSDORead);
	EplSDORead(&EPLInverter[3].fub.fnEplSDORead);

	EplSDOWrite(&EPLInverter[0].fub.fnEplSDOWrite);
	EplSDOWrite(&EPLInverter[1].fub.fnEplSDOWrite);
	EplSDOWrite(&EPLInverter[2].fub.fnEplSDOWrite);
	EplSDOWrite(&EPLInverter[3].fub.fnEplSDOWrite);

}

void _EXIT eplExit(void)
{
	// Insert code here

}
```

#### epl.typ - Local data types
```iecst
TYPE
	epl_typ : 	STRUCT  (*datatype for AsEPL Library*)
		cmd : eplCmd_typ; (*variable with commands*)
		para : eplPara_typ; (*variable with parameters*)
		fub : eplFUB_typ; (*variable with Function Blocks*)
		state : state_enum; (*variable with actual state*)
	END_STRUCT;
	eplCmd_typ : 	STRUCT  (*datatype with commands*)
		readNode : BOOL; (*command to read the Node Number of the Powerlink interface*)
		readThresholdCnt : BOOL; (*command to read an Object Entry*)
		index : UINT;
		subindex : USINT;
		bWriteObj : BOOL;
		bReadObj : BOOL;
	END_STRUCT;
	eplPara_typ : 	STRUCT  (*datatype with parameters*)
		nodeNr : USINT; (*Node number of the Powerling interface*)
		readData : UDINT; (*Read Data*)
		writeData : UDINT; (*Data to be written*)
		MotorVoltage : UINT; (*Motor voltage from parameter read*)
		MotorPower : INT; (*Motor power from parameter read*)
		EnergyCons : UINT;
	END_STRUCT;
	eplFUB_typ : 	STRUCT  (*datatype with Function Blocks*)
		fnEplGetLocalNodeID : EplGetLocalNodeID; (*FUB to get Node Number of local Powerlink interface*)
		fnEplSDOWrite : EplSDOWrite; (*FUB to write a node's object entries*)
		fnEplSDORead : EplSDORead; (*FUB to read a node's object entries*)
	END_STRUCT;
	state_enum :
		( (*enumerators for the state in the task*)
		EPL_WAIT, (*state to wait for any commands*)
		EPL_READ_NODE, (*state to read powerlink node number*)
		EPL_READ_OE, (*state to read object entry*)
		EPL_WRITE_OE, (*state to write object entry*)
		EPL_ERROR (*state when an error occured*)
		);
END_TYPE
```

#### epl.var - Local variables
```iecst
(*Powerlink Read/Write Function*)
VAR
	EPLInverter : ARRAY[0..3] OF epl_typ;
END_VAR
(*Variable*)
VAR
	uIndexRead : ARRAY[0..3] OF USINT; (*Index of regester for read*)
	uIndexExtru : USINT;
	sDevice : ARRAY[0..3] OF STRING[80];
	uIndexOffset : USINT;
	bTestRead : BOOL;
	sDeviceAExtr : STRING[80];
	i : USINT;
END_VAR
(*Power Consumption*)
VAR
	rActCurrentA : ARRAY[0..59] OF REAL;
	rActCurrentB : ARRAY[0..59] OF REAL;
	rActCurrentC : ARRAY[0..59] OF REAL;
	rActCurrentV : ARRAY[0..59] OF REAL;
	rActVoltageA : ARRAY[0..59] OF REAL;
	rActVoltageB : ARRAY[0..59] OF REAL;
	rActVoltageC : ARRAY[0..59] OF REAL;
	rActVoltageV : ARRAY[0..59] OF REAL;
	rPowerA : ARRAY[0..59] OF REAL;
	rPowerTotalPerSecA : REAL;
	rPowerPerSecA : REAL;
	uStepPowerA : UDINT;
	uCountTimerA : UDINT;
	uIndexA : UDINT;
	bCleanPowerA : BOOL;
	iClickTimeA : INT;
END_VAR
VAR RETAIN
	rPowerTotalA : REAL;
	rPowerPerHrA : REAL;
END_VAR
VAR
	rPowerB : ARRAY[0..59] OF REAL;
	rPowerTotalPerSecB : REAL;
	rPowerPerSecB : REAL;
	uStepPowerB : UDINT;
	uCountTimerB : UDINT;
	uIndexB : UDINT;
	bCleanPowerB : BOOL;
	iClickTimeB : INT;
END_VAR
VAR RETAIN
	rPowerTotalB : REAL;
	rPowerPerHrB : REAL;
END_VAR
VAR
	rPowerC : ARRAY[0..59] OF REAL;
	rPowerTotalPerSecC : REAL;
	rPowerPerSecC : REAL;
	uStepPowerC : UDINT;
	uCountTimerC : UDINT;
	uIndexC : UDINT;
	bCleanPowerC : BOOL;
	iClickTimeC : INT;
END_VAR
VAR RETAIN
	rPowerTotalC : REAL;
	rPowerPerHrC : REAL;
END_VAR
VAR
	rPowerV : ARRAY[0..59] OF REAL;
	rPowerTotalPerSecV : REAL;
	rPowerPerSecV : REAL;
	uStepPowerV : UDINT;
	uCountTimerV : UDINT;
	uIndexV : UDINT;
	bCleanPowerV : BOOL;
	iClickTimeV : INT;
END_VAR
VAR RETAIN
	rPowerTotalV : REAL;
	rPowerPerHrV : REAL;
END_VAR
VAR
	fnTON_10msA : TON_10ms;
	fnTON_10msB : TON_10ms;
	fnTON_10msC : TON_10ms;
	fnTON_10msV : TON_10ms;
	i_A : UINT;
	i_B : UINT;
	i_C : UINT;
	i_V : UINT;
	fnTON_10msA_HR : TON_10ms;
	fnTON_10msB_HR : TON_10ms;
	fnTON_10msC_HR : TON_10ms;
	fnTON_10msV_HR : TON_10ms;
	uStepPowerHourA : UDINT;
	uStepPowerHourB : UDINT;
	uStepPowerHourC : UDINT;
	uStepPowerHourV : UDINT;
	bTestAuto : BOOL;
	rPowerPerMinA : REAL;
	rPowerPerMinB : REAL;
	rPowerPerMinC : REAL;
	rPowerPerMinV : REAL;
	rTestVoltage : REAL;
	rTestCurrent : REAL;
END_VAR
```

### Package Logical/log_info - PLC system log information

### Program Logical/log_info/loginfo (ANSIC, version 1.00.0) - system log infomation

- pic_id.h (reference to Logical/GlobalIncludes/pic_id.h)

#### loginfo.c
```c
/**************************************************************************************
*   Copyright:  2010  BERNECKER & RAINER Industrie-Elektronik Ges.m.b.H       															*
*-------------------------------------------------------------------------------------*
*        Identification:                                                              *
*       Taskname : loginfo                                                            *
*       Filename : loginfo.c                                                          *
*       Description : plc log information                                             *
*-------------------------------------------------------------------------------------*
*   History                                                                           *
*   Version     Date         Autor                                                    *
*   01.00       2010.10.8    B&R China     created                       	          *
*   CmdPageUp    -----  system log page up                                     		  *
*   CmdPageDown  -----  system log page down                                          *
*   OptionLog    -----  change log type                                               *
**************************************************************************************/

#include <bur/plctypes.h>
#include <string.h>

#ifdef _DEFAULT_INCLUDES
#include <AsDefault.h>
#endif

#include "pic_id.h"

/***************************************************************************************
**                              define                                                **
***************************************************************************************/
#define 	C_MAX_LOG_BUFFER      27
#define 	C_MAX_LOG_SCREEN      25

/***************************************************************************************
**                            defines                                                 **
***************************************************************************************/
#define		STEP_WAIT			 0
#define		STEP_GET_INFO		10
#define		STEP_READ_INIT		20
#define		STEP_READ		  	30
#define		STEP_ERR_CHECK	    40
#define		STEP_GET_TEXT		50
#define		STEP_READ_ADD		60
#define		STEP_READ_END		70
#define		STEP_READ_ERR		999

/**************************************************************************************/
/*   						  Functions					                              */
/**************************************************************************************/

/**************************************************************************************
****                    I N I T U P  O F   T H E   T A S K                         ****
**************************************************************************************/
_INIT void init ()
{
	DOInfo.enable = 1;
 	DOInfo.pName  = (UDINT) "log_txt";
    DatObjInfo(&DOInfo);
 	if (DOInfo.status == 0) /* Data object not found or error -> Just don't copy the error message */
	{
		doIdent = DOInfo.ident;
		pSrc = (SINT *)DOInfo.pDatObjMem;
	}
	else
	{
	    pSrc = 0;
	}

	bCmdRefresh = 1;
	OptionLog  = arlogLEVEL_FATAL - 1;  /* error log   */
	StepLog = STEP_WAIT;

	actualIndexOld = 0;
}/* End of Init */
/**************************************************************************************
****                C Y C L I C   P A R T   O F   T H E   T A S K                  ****
**************************************************************************************/
_CYCLIC void cyclic ()
{
	STRING strTemp[30];
	/* page change to system log page */
	if(gPanelObj.GetPicture == PIC_LOG_INFO && oldPicture != PIC_LOG_INFO)
	{
		bCmdRefresh = 1;
	}
	oldPicture = gPanelObj.GetPicture;

	/* ----------------- log type change ----------------- */
	if(OptionLog != OptionLogOld)
	{
		bCmdRefresh    = 1;
		bCmdTypeChange = 1;
	}

	OptionLogOld = OptionLog;

	/* ----------------- step mathine control ----------------- */
	switch(StepLog)
	{
		case STEP_WAIT:
			if(1 == bCmdRefresh)
			{
				bCmdRefresh = 0;
				StepLog = STEP_GET_INFO;
			}

			if(1 == bCmdPageDown)
			{
				bCmdPageDown = 0;
				if(indexRecord > 0)
				{
					StepLog = STEP_READ_INIT;
				}
			}
			else if(1 == bCmdPageUp)
			{
				bCmdPageUp = 0;
				if(indexRecord + C_MAX_LOG_SCREEN <= AsArLogGetInfo_0.actualIndex)
				{
					indexRecord = indexRecord + C_MAX_LOG_SCREEN;
					StepLog = STEP_READ_INIT;
				}
			}
			else if(1 == bCmdPageInit)
			{
				bCmdPageInit = 0;
				indexRecord = AsArLogGetInfo_0.actualIndex;

				StepLog = STEP_READ_INIT;
			}
			else if(1 == bCmdPageEnd)
			{
				bCmdPageEnd = 0;

				if(AsArLogGetInfo_0.actualIndex >= C_MAX_LOG_SCREEN)
				{
					indexRecord = C_MAX_LOG_SCREEN;
				}
				else
				{
					indexRecord = AsArLogGetInfo_0.actualIndex;
				}
			}
			break;

		case STEP_GET_INFO:
			AsArLogGetInfo_0.enable = 1;
			AsArLogGetInfo_0.ident = arlogBASE_SYSTEM_LOG_IDENT;

			/* call function  */
			AsArLogGetInfo(&AsArLogGetInfo_0);

			if(AsArLogGetInfo_0.status != ERR_OK )
			{
				if(AsArLogGetInfo_0.status == ERR_FUB_BUSY)
				{
					AsArLogGetInfo_0.enable = 1;
				}
				else
				{
					AsArLogGetInfo_0.enable = 0;
					StepLog = STEP_READ_ERR;
				}
			}
			else
			{
				AsArLogGetInfo_0.enable = 0;

				if(0 == bCmdTypeChange)
				{
					if(actualIndexOld != AsArLogGetInfo_0.actualIndex)
					{
						actualIndexOld = AsArLogGetInfo_0.actualIndex;
						indexRecord = AsArLogGetInfo_0.actualIndex;
						StepLog = STEP_READ_INIT;
					}
					else
					{
						StepLog = STEP_WAIT;
					}
				}
				else
				{
					bCmdTypeChange = 0;
					actualIndexOld = AsArLogGetInfo_0.actualIndex;
					indexRecord = AsArLogGetInfo_0.actualIndex;
					StepLog = STEP_READ_INIT;
				}
			}
			break;

		case STEP_READ_INIT:
			percentProgressBar = 0;
			indexLog = 0;
			memset(&LogBuffer,0,sizeof(LogBuffer));
			memset(&LogDataOld,0,sizeof(LogDataOld));
			strcpy(sLogContext,"");
			StepLog = STEP_READ;
			break;

		case STEP_READ:
			AsArLogRead_0.enable = 1;
			AsArLogRead_0.ident  = AsArLogGetInfo_0.ident;
			AsArLogRead_0.index  = indexRecord;
			AsArLogRead_0.arlogRead = (UDINT)&LogData;
			AsArLogRead_0.memBin  = (UDINT)&LogBin;
			AsArLogRead_0.lenBin  = 100;
			AsArLogRead_0.memAscii  = (UDINT)&sLogContext;
			AsArLogRead_0.lenAscii  = 100;

			/* call function  */
			AsArLogRead(&AsArLogRead_0);

			if(AsArLogRead_0.status != ERR_OK && AsArLogRead_0.status != arlogERR_READ_BINARY_BUFFER)
			{
				if(AsArLogRead_0.status == ERR_FUB_BUSY)
				{
					AsArLogRead_0.enable = 1;
				}
				else
				{
					AsArLogRead_0.enable = 0;
					StepLog = STEP_READ_ERR;
				}
			}
			else /* if(AsArLogRead_0.status != ERR_OK) */
			{
				AsArLogRead_0.enable = 0;

				/* compact logbook from pcc and display  */
				if(LogData.errornr == LogDataOld.errornr  && LogData.errDay == LogDataOld.errDay  &&
					LogData.errHour == LogDataOld.errHour  && LogData.errMinute == LogDataOld.errMinute)
				{
					StepLog = STEP_READ_ADD;	/* skip  */
				}/*  if(A && B && C	&& D && E) */
				else
				{
					if( LogData.logLevel == OptionLog + 1 )
					{
						/* error number  */
						itoa((DINT)LogData.errornr, (UDINT)sTmp);
						strcat(LogBuffer.strErrNr[indexLog], sTmp);

						/* error task name  */
						memcpy(strTemp,LogData.taskName,30);
						strcpy(LogBuffer.strTaskName[indexLog],strTemp);

						/* get error occur time to string  */
						strcpy(LogBuffer.strTime[indexLog], "");

						itoa((DINT)LogData.errYear, (UDINT)sTmp);
						strcat(LogBuffer.strTime[indexLog], sTmp);

						strcat(LogBuffer.strTime[indexLog], "/");
						if(LogData.errMonth<10)strcat(LogBuffer.strTime[indexLog], "0");
						itoa((DINT)LogData.errMonth, (UDINT)sTmp);
						strcat(LogBuffer.strTime[indexLog], sTmp);

						strcat(LogBuffer.strTime[indexLog], "/");
						if(LogData.errDay<10)strcat(LogBuffer.strTime[indexLog], "0");
						itoa((DINT)LogData.errDay, (UDINT)sTmp);
						strcat(LogBuffer.strTime[indexLog], sTmp);

						strcat(LogBuffer.strTime[indexLog], " ");
						if(LogData.errHour<10)strcat(LogBuffer.strTime[indexLog], "0");
						itoa((DINT)LogData.errHour, (UDINT)sTmp);
						strcat(LogBuffer.strTime[indexLog], sTmp);

						strcat(LogBuffer.strTime[indexLog], ":");
						if(LogData.errMinute<10)strcat(LogBuffer.strTime[indexLog], "0");
						itoa((DINT)LogData.errMinute, (UDINT)sTmp);
						strcat(LogBuffer.strTime[indexLog], sTmp);

						strcat(LogBuffer.strTime[indexLog], ":");
						if(LogData.errSecond<10)strcat(LogBuffer.strTime[indexLog], "0");
						itoa((DINT)LogData.errSecond, (UDINT)sTmp);
						strcat(LogBuffer.strTime[indexLog], sTmp);

						LogDataOld = LogData;
						if(strlen(sLogContext) == 0)
						{
							StepLog = STEP_ERR_CHECK;
						}
						else
						{
							strcpy(LogBuffer.strContext[indexLog], sLogContext);
							indexLog = indexLog+1;
							StepLog = STEP_READ_ADD;
						}
					}/* if( LogData.logLevel == OptionLog + 1) */
					else
					{
						StepLog = STEP_READ_ADD;
					}
				}/*  if(A && B && C	&& D && E)else */
			}/* if(AsArLogRead_0.status != ERR_OK) */
			break;

		case STEP_ERR_CHECK:
			if((DOInfo.status == 0)&&(pDat != 0))
			{
				pDat = pSrc;
				StepLog = STEP_GET_TEXT;
			}
			else
			{
				strcpy(LogBuffer.strContext[indexLog], "Can not find,please find out in help");
				StepLog = STEP_READ_ADD;
			}
			break;

		case STEP_GET_TEXT:
			do
			{
				/* Copy the error number */
				if(LogData.errornr <= 65535)  /* ERROR NUBER IS UINT */
				{
					memcpy(&error_read,pDat,2);
					pDat++;
					pDat++;   /* " */
				}
				else                         /* ERROR NUBER IS UDINT */
				{
					memcpy(&error_read,pDat,4);
					pDat++;
					pDat++;
					pDat++;
					pDat++;	/* " */
				}
				if(error_read == LogData.errornr)				/* The index error is founded */
				{
					strcpy(LogBuffer.strContext[indexLog],pDat);/* Copy the error string      */
					break;
				}
				else if(error_read > LogData.errornr)
				{
					strcpy(LogBuffer.strContext[indexLog],"The error string is not in the data base!");
					break;
				}

				while(*pDat != 0) pDat++;		/* Find the end of the string */
				pDat++;							/* Go to the start of the error number */
			}while(pDat <= ((SINT *) DOInfo.pDatObjMem + DOInfo.len));
			indexLog = indexLog+1;
			StepLog = STEP_READ_ADD;
			break;

		case STEP_READ_ADD:
			strcpy(sLogContext,"");
			indexRecord--;

			if((indexRecord == 0) || (indexLog == C_MAX_LOG_BUFFER))
			{
				StepLog = STEP_READ_END;
			}
			else
			{
				StepLog = STEP_READ;
			}
			break;

		case STEP_READ_END:
			StepLog = STEP_WAIT;
			break;

		case STEP_READ_ERR:
			AsArLogGetInfo_0.enable = 0;
			AsArLogRead_0.enable    = 0;
			StepLog = STEP_WAIT;
			break;

		default:
			break;
	}/* switch(StepLog) */

	/* ------------ progress bar display ------------ */
	if(StepLog > STEP_READ_INIT && StepLog < STEP_READ_END)
	{

		if(OptionLog != arlogLEVEL_WARNING - 1) /* warnning  */
		{
			if(AsArLogGetInfo_0.actualIndex > 0)
			{
				percentProgressBar = (AsArLogGetInfo_0.actualIndex - indexRecord) * 100/AsArLogGetInfo_0.actualIndex ;
			}
		}
		else									/*    */
		{
			if(AsArLogGetInfo_0.actualIndex > C_MAX_LOG_SCREEN)
			{
				percentProgressBar = indexLog * 4;
			}
			else if(AsArLogGetInfo_0.actualIndex > 1)
			{
				percentProgressBar = indexLog * 100 / (AsArLogGetInfo_0.actualIndex-1) ;
			}
		}
	}/* if(StepLog > C_STEP_READ_INIT && StepLog < C_STEP_READ_END) */
}/* End of cyclic */
```

#### loginfo.typ - variable data types
```iecst
(********************************************************************
 * COPYRIGHT --
 ********************************************************************
 * Package: log_info
 * File: log_info.typ
 * Author: lij
 * Created: July 02, 2012
 ********************************************************************
 * Data types of package log_info
 ********************************************************************)

TYPE
	Log_Buffer_typ : 	STRUCT
		strTime : ARRAY[0..MAX_LOG_BUFFER]OF STRING[79];
		strTaskName : ARRAY[0..MAX_LOG_BUFFER]OF STRING[31];
		strErrNr : ARRAY[0..MAX_LOG_BUFFER]OF STRING[5];
		strContext : ARRAY[0..MAX_LOG_BUFFER]OF STRING[119];
	END_STRUCT;
END_TYPE
```

#### loginfo.var
```iecst
VAR
	StepLog : UINT;
	LogBuffer : Log_Buffer_typ;
	indexLog : UINT;
	indexRecord : UINT;
	AsArLogGetInfo_0 : AsArLogGetInfo;
	AsArLogRead_0 : AsArLogRead;
	LogData : asarlogRead;
	sLogContext : STRING[119];
	sTmp : STRING[79];
	DOInfo : DatObjInfo;
	doIdent : UDINT;
	error_read : UDINT;
	LogBin : ARRAY[0..119] OF SINT;
	actualIndexOld : UDINT;
	bCmdRefresh : BOOL;
	OptionLog : USINT;
	percentProgressBar : UINT;
	OptionLogOld : USINT;
	LogDataOld : asarlogRead;
	pSrc : REFERENCE TO SINT;
	pDat : REFERENCE TO SINT;
	oldPicture : UINT;
	bCmdTypeChange : BOOL;
	bCmdPageDown : BOOL;
	bCmdPageUp : BOOL;
	bCmdPageInit : BOOL;
	bCmdPageEnd : BOOL;
END_VAR
```

### Data object Logical/log_info/log_txt (Simple, version 3.09.0) - Data index of the logbook error

- log_txt.dat (not shown)

### Package Logical/VarChgLog - point var change log info

### Program Logical/VarChgLog/pvchg (ANSIC, version 1.00.0) - variable change log

#### pvchg.c
```c
/********************************************************************
 * COPYRIGHT --  B&R China
 ********************************************************************
 * Program: pvchg
 * File: pvchg.c
 * Author: lijianjun
 * Created: March 06, 2013
 ********************************************************************
 * Implementation of program pvchg --- point variable change logger
 ********************************************************************/

#include <bur/plctypes.h>
#include <string.h>

#ifdef _DEFAULT_INCLUDES
#include <AsDefault.h>
#endif

#include "keyap2100.h"
#include "pic_id.h"
#include "edge.h"

/*********************************************************************
**                            defines                               **
*********************************************************************/
#define		C_STEP_WAIT			     100
#define		C_STEP_SAVE		         1000
#define		C_STEP_LOAD			     2000
#define		C_STEP_ERR_CHECK	     3000

#define 	S$UNIT_LENGTH		      8
#define		S$LINE_LENGTH		      (C_PV_NAME_LENGTH + 1 + 4)

#define		S$LOG_MAX_NO	         200
#define     S$LOG_MAX_SCREEN        (C_MAX_LOG__SCREEN + 1)

/**************************************************************************************
**                            Function Declarations								     **
**************************************************************************************/
void fun_pv_name();

/**************************************************************************************
**     	        		I N I T U P  O F   T H E   T A S K 		 				     **
**************************************************************************************/
_INIT void pvchg_init(void)
{
	memset(VarInfoList,0,sizeof(VarInfoList));
	strcpy(pv_get.modname,"pv_chg");

	strcpy(DataObjOperate.ModName,"pvchglog");

	DataObjOperate.InitStep = 100;
	DataObjOperate.Step = C_STEP_WAIT;

	pvChange = 0;

}/* end of _INIT */

/*************************************************************************************
**        				C Y C L I C   P A R T   O F   T H E   T A S K  				**
*************************************************************************************/
_CYCLIC void pvchg_cyc(void)
{
	gMachinePara.MoldL.Carriage.V_Bw = gMachinePara.MoldL.Carriage.V_Bw;

	int idx, buffer_idx;

	/* ---------------- step machine init ---------------- */
	switch(DataObjOperate.InitStep)
	{
		case 100:
			fun_pv_name ();
			if (pv_get.errorNum != 0)
			{
				DataObjOperate.InitStep = 9999;
			}
			else
			{
				pv_get.length = DOInfo.len;
				DataObjOperate.Ident  = DOInfo.ident;
				DataObjOperate.InitStep = 200;
			}
			break;

		case 200:
			DOInfo.enable	= 1;
			DOInfo.pName	= (UDINT)DataObjOperate.ModName;
			/* Call  FUB  */
			DatObjInfo(&DOInfo);
			if (DOInfo.status == doERR_MODULNOTFOUND)	/* Data module not found -> create a new one */
			{
				DataObjOperate.InitStep  = 300;
			}
			else
			{
				DataObjOperate.Ident  = DOInfo.ident;
				DataObjOperate.InitStep = 900;
			}
			break;

		case 300:
			/* Initialize create structure */
			DOCreate.enable 	= 1;
			DOCreate.grp	 	= 0;
			DOCreate.pName 	= (UDINT)DataObjOperate.ModName;
			DOCreate.len 		= sizeof(VarLog) * (S$LOG_MAX_NO + 1) + 4;
				DOCreate.MemType 	= doUSRROM;
			DOCreate.Option 	= 0;
			DOCreate.pCpyData 	= 0;
			/* Call FUB */
			DatObjCreate(&DOCreate);
			/* Get FUB output information */
			if( 0 == DOCreate.status)
			{
				idxLog = 0;
				DOCreate.enable = 0;
				DataObjOperate.Ident    = DOCreate.ident;
				DataObjOperate.InitStep = 1000;
			}
			break;

		case 400:
			status_tmpalloc = TMP_alloc(sizeof(VarLog) * (S$LOG_MAX_NO + 1) + 4,(void**)&pData);
				if(0 == status_tmpalloc)
			{
				memset(pData,0,sizeof(VarLog) * (S$LOG_MAX_NO + 1) + 4);
					DataObjOperate.InitStep = 500;
			}
			else
			{
				DataObjOperate.InitStep = 9999;
			}
			break;

		case 500:
			DOWrite.enable  = 1;
			DOWrite.ident   = DataObjOperate.Ident;
			DOWrite.Offset  = 0;
			DOWrite.pSource = (UDINT)pData;
			DOWrite.len 	= sizeof(VarLog) * (S$LOG_MAX_NO + 1) + 4;

				/* Call FUB */
				DatObjWrite(&DOWrite);

			if(0 == DOWrite.status)
			{
				DOWrite.enable = 0;
				DataObjOperate.InitStep = 600;
			}
			break;

		case 600:
			status_tmpfree = TMP_free(sizeof(VarLog) * (S$LOG_MAX_NO + 1) + 4,(void**)pData);
				if(0 == status_tmpfree)
			{
				idxLog = 0;
				idxScreen = 0;
				memset(&VarLogList[0],0,sizeof(VarLogList));
				memset(&VarNameList[0],0,sizeof(VarNameList));

				memset(&VarLogList_Buffer[0],0,sizeof(VarLogList_Buffer));
				memset(&VarNameList_Buffer[0],0,sizeof(VarNameList_Buffer));

				DataObjOperate.InitStep = 1000;
			}
			else
			{
				DataObjOperate.InitStep = 9999;
			}
			break;

		case 900:
			DORead.enable 		= 1;
			DORead.ident 		= DataObjOperate.Ident;
			DORead.Offset 		= 0;
			DORead.pDestination	= (UDINT)(&idxLog);
			DORead.len 			= sizeof(idxLog);

			/* Call FUB */
			DatObjRead(&DORead);

			/* Get status */
			if(0 == DORead.status)
			{
				DORead.enable = 0;
				DataObjOperate.InitStep = 1000;
			}
			break;

		case 1000:
			DataObjOperate.InitStep = 3000;
			break;

		case 9999:

			break;
	}/* switch(DataObjOperate.InitStep) */

	if(DOInfo.ident == 0 || DataObjOperate.InitStep != 3000)
	{
		return;
	}
	else
	{
		/* GET pv change edge */
		for(idx=0; idx<pv_get.length/S$LINE_LENGTH;idx++)
			{
			switch ((unsigned short)(VarInfoList[idx].typ))
			{
				/******* BIT *******/
				case 1:
					if( (*((plcbit *)VarInfoList[idx].address)) != (*((plcbit *)VarInfoList[idx].pValue)) )
					{
						pvChange = 1;
						VarLog.idxGroup = VarInfoList[idx].idxGroup;
						VarLog.idxText = VarInfoList[idx].idxText;
						strcpy(VarLog.chgTime,gPanelObj.CurrentTime);
						itoa((DINT)(*((plcbit *)VarInfoList[idx].pValue)),(UDINT)VarLog.oldValue);
						itoa((DINT)(*((plcbit *)VarInfoList[idx].address)),(UDINT)VarLog.curValue);
					}
					(*((plcbit *)VarInfoList[idx].pValue)) = (*((plcbit *)VarInfoList[idx].address));
					break;

				/******* INT8 *******/
				case 2:
					if( (*((SINT *)VarInfoList[idx].address)) != (*((SINT *)VarInfoList[idx].pValue)) )
					{
						pvChange = 1;
						VarLog.idxGroup = VarInfoList[idx].idxGroup;
						VarLog.idxText = VarInfoList[idx].idxText;
						strcpy(VarLog.chgTime,gPanelObj.CurrentTime);
						itoa((DINT)(*((SINT *)VarInfoList[idx].pValue)),(UDINT)VarLog.oldValue);
						itoa((DINT)(*((SINT *)VarInfoList[idx].address)),(UDINT)VarLog.curValue);
					}
					(*((SINT *)VarInfoList[idx].pValue)) = (*((SINT *)VarInfoList[idx].address));

					break;

				/******* INT16 *******/
				case 3:
					if( (*((INT *)VarInfoList[idx].address)) != (*((INT *)VarInfoList[idx].pValue)) )
					{
						pvChange = 1;
						VarLog.idxGroup = VarInfoList[idx].idxGroup;
						VarLog.idxText = VarInfoList[idx].idxText;
						strcpy(VarLog.chgTime,gPanelObj.CurrentTime);
						itoa((DINT)(*((INT *)VarInfoList[idx].pValue)),(UDINT)VarLog.oldValue);
						itoa((DINT)(*((INT *)VarInfoList[idx].address)),(UDINT)VarLog.curValue);
					}
					(*((INT *)VarInfoList[idx].pValue)) = (*((INT *)VarInfoList[idx].address));

					break;

				/******* INT32 *******/
				case 4:
					if( (*((DINT *)VarInfoList[idx].address)) != (*((DINT  *)VarInfoList[idx].pValue)) )
					{
						pvChange = 1;
						VarLog.idxGroup = VarInfoList[idx].idxGroup;
						VarLog.idxText = VarInfoList[idx].idxText;
						strcpy(VarLog.chgTime,gPanelObj.CurrentTime);
						itoa((DINT)(*((INT *)VarInfoList[idx].pValue)),(UDINT)VarLog.oldValue);
						itoa((DINT)(*((INT *)VarInfoList[idx].address)),(UDINT)VarLog.curValue);
					}
					(*((DINT *)VarInfoList[idx].pValue)) = (*((DINT *)VarInfoList[idx].address));

					break;

				/******* BYTE *******/
				case 5:
					if( (*((USINT *)VarInfoList[idx].address)) != (*((USINT *)VarInfoList[idx].pValue)) )
					{
						pvChange = 1;
						VarLog.idxGroup = VarInfoList[idx].idxGroup;
						VarLog.idxText = VarInfoList[idx].idxText;
						strcpy(VarLog.chgTime,gPanelObj.CurrentTime);
						itoa((DINT)(*((USINT *)VarInfoList[idx].pValue)),(UDINT)VarLog.oldValue);
						itoa((DINT)(*((USINT *)VarInfoList[idx].address)),(UDINT)VarLog.curValue);
					}
					(*((USINT *)VarInfoList[idx].pValue)) = (*((USINT *)VarInfoList[idx].address));

					break;

				/******* WORD *******/
				case 6:
					if( (*((UINT *)VarInfoList[idx].address)) != (*((UINT *)VarInfoList[idx].pValue)) )
					{
						pvChange = 1;
						VarLog.idxGroup = VarInfoList[idx].idxGroup;
						VarLog.idxText = VarInfoList[idx].idxText;
						strcpy(VarLog.chgTime,gPanelObj.CurrentTime);
						itoa((DINT)(*((UINT *)VarInfoList[idx].pValue)),(UDINT)VarLog.oldValue);
						itoa((DINT)(*((UINT *)VarInfoList[idx].address)),(UDINT)VarLog.curValue);
					}
					(*((UINT *)VarInfoList[idx].pValue)) = (*((UINT *)VarInfoList[idx].address));

					break;

				/******* LONG *******/
				case 7:
					if( (*((UDINT *)VarInfoList[idx].address)) != (*((UDINT *)VarInfoList[idx].pValue)) )
					{
						pvChange = 1;
						VarLog.idxGroup = VarInfoList[idx].idxGroup;
						VarLog.idxText = VarInfoList[idx].idxText;
						strcpy(VarLog.chgTime,gPanelObj.CurrentTime);
						itoa((DINT)(*((UDINT *)VarInfoList[idx].pValue)),(UDINT)VarLog.oldValue);
						itoa((DINT)(*((UDINT *)VarInfoList[idx].address)),(UDINT)VarLog.curValue);

					}
					(*((UDINT *)VarInfoList[idx].pValue)) = (*((UDINT *)VarInfoList[idx].address));
					break;

				/******* FLOAT *******/
				case 8:
					if( (*((REAL *)VarInfoList[idx].address)) != (*((REAL *)VarInfoList[idx].pValue)) )
					{
						pvChange = 1;
						VarLog.idxGroup = VarInfoList[idx].idxGroup;
						VarLog.idxText = VarInfoList[idx].idxText;
						strcpy(VarLog.chgTime,gPanelObj.CurrentTime);
						ftoa((*((REAL *)VarInfoList[idx].pValue)),(UDINT)VarLog.oldValue);
						ftoa((*((REAL *)VarInfoList[idx].address)),(UDINT)VarLog.curValue);
					}
					(*((REAL *)VarInfoList[idx].pValue)) = (*((REAL *)VarInfoList[idx].address));
					break;

				default:
					break;
			}/* End of switch */
		}/* for(idx=0; idx<DOInfo.len/S$LINE_LENGTH,idx++) */

		/* step machine save and load  */
		switch (DataObjOperate.Step)
		{
			case C_STEP_WAIT:
				if(1 == pvChange)
				{
					pvChange = 0;
					DataObjOperate.Step = C_STEP_SAVE;
				}

				if(oldIdxLog  != idxLog)
				{
					memset(&VarLogList[0],0,sizeof(VarLogList));
					memset(&VarNameList[0],0,sizeof(VarNameList));

					memset(&VarLogList_Buffer[0],0,sizeof(VarLogList_Buffer));
					memset(&VarNameList_Buffer[0],0,sizeof(VarNameList_Buffer));

					//					idxScreen = ((idxLog/S$LOG_MAX_SCREEN  * S$LOG_MAX_SCREEN )%S$LOG_MAX_NO);

					//					idxScreen = 0;
					DataObjOperate.Step = C_STEP_LOAD;
					oldIdxLog  = idxLog;
				}

				if(gPanelObj.GetPicture == PIC_PV_LOG)
				{
					CmdPageUp 	= EDGEPOS(gPanelObj.KeyMatric[S$KEYMATRIX_F6],OldF6);
					CmdPageDown = EDGEPOS(gPanelObj.KeyMatric[S$KEYMATRIX_F7],OldF7);

					if(1 == CmdDelete)
					{
						CmdDelete = 0;
						DataObjOperate.InitStep = 400;
					}
					else if(1 == CmdPageUp)
					{
						CmdPageUp = 0;
						memset(&VarLogList[0],0,sizeof(VarLogList));
						memset(&VarNameList[0],0,sizeof(VarNameList));

						memset(&VarLogList_Buffer[0],0,sizeof(VarLogList_Buffer));
						memset(&VarNameList_Buffer[0],0,sizeof(VarNameList_Buffer));

						if(idxScreen >= S$LOG_MAX_SCREEN)idxScreen = idxScreen - S$LOG_MAX_SCREEN;
						DataObjOperate.Step = C_STEP_LOAD;
					}
					else if(1 == CmdPageDown)
					{
						if(idxLog >= S$LOG_MAX_SCREEN)
						{
							CmdPageDown = 0;
							memset(&VarLogList[0],0,sizeof(VarLogList));
							memset(&VarNameList[0],0,sizeof(VarNameList));

							memset(&VarLogList_Buffer[0],0,sizeof(VarLogList_Buffer));
							memset(&VarNameList_Buffer[0],0,sizeof(VarNameList_Buffer));

							if(idxScreen < S$LOG_MAX_NO - S$LOG_MAX_SCREEN)idxScreen = idxScreen + S$LOG_MAX_SCREEN;

							DataObjOperate.Step = C_STEP_LOAD;
						}
					}
					else if(1 == bRefresh)
					{
						bRefresh = 0;
						memset(&VarLogList[0],0,sizeof(VarLogList));
						memset(&VarNameList[0],0,sizeof(VarNameList));

						memset(&VarLogList_Buffer[0],0,sizeof(VarLogList_Buffer));
						memset(&VarNameList_Buffer[0],0,sizeof(VarNameList_Buffer));
						DataObjOperate.Step = C_STEP_LOAD;
					}
				}
				else
				{
					bRefresh = 1;
				}

				break;

			/* ---------------- Save to data module ---------------- */
			case C_STEP_SAVE:
				DOWrite.enable 	= 1;
				DOWrite.ident 	= DataObjOperate.Ident;
				DOWrite.Offset 	= sizeof(VarLog) * (idxLog %S$LOG_MAX_NO) + sizeof(idxLog);
					DOWrite.pSource = (UDINT)(&VarLog);
				DOWrite.len     = sizeof(VarLog);

				DatObjWrite(&DOWrite);

				if(0 == DOWrite.status)
				{
					DOWrite.enable = 0;
					DataObjOperate.Step = C_STEP_SAVE + 100;
				}
				break;

			case C_STEP_SAVE + 100:
				idxLog = idxLog + 1;
				if(idxLog == S$LOG_MAX_NO-1)
					{
					idxLog = 0;
					CmdDelete = 1;
					DataObjOperate.Step = C_STEP_WAIT;
				}
				else
				{
					DataObjOperate.Step = C_STEP_SAVE + 200;
				}
				break;

			case C_STEP_SAVE + 200:
				DOWrite.enable 	= 1;
				DOWrite.ident 	= DataObjOperate.Ident;
				DOWrite.Offset 	= 0;
				DOWrite.pSource = (UDINT)(&idxLog);
				DOWrite.len     = sizeof(idxLog);

				DatObjWrite(&DOWrite);

				if(0 == DOWrite.status)
				{
					DOWrite.enable = 0;
					DataObjOperate.Step = C_STEP_SAVE + 300;
				}
				break;

			case C_STEP_SAVE + 300:
				DataObjOperate.Step = C_STEP_WAIT;
				break;

			/* ---------------- read from data module ---------------- */
			case C_STEP_LOAD:
				DORead.enable 		= 1;
				DORead.ident 		= DataObjOperate.Ident;
				if(0 == idxScreen)
				{
					if(idxLog < S$LOG_MAX_SCREEN)
					{
						DORead.Offset = 0* sizeof(VarLog) + sizeof(idxLog);
					}
					else
					{
						DORead.Offset = (idxLog-S$LOG_MAX_SCREEN)* sizeof(VarLog) + sizeof(idxLog);
					}
				}
				else  //page change
				{
					if((idxLog - idxScreen) < idxScreen)
					{
						DORead.Offset = 0* sizeof(VarLog) + sizeof(idxLog);
					}
					else
					{
						DORead.Offset = (idxLog-idxScreen*2)* sizeof(VarLog) + sizeof(idxLog);
					}

				}
				DORead.pDestination	= (UDINT)(&VarLogList_Buffer[0]);
				DORead.len 			= sizeof(VarLogList_Buffer);

				/* Call FUB */
				DatObjRead(&DORead);

				/* Get status */
				if(0 == DORead.status)
				{
					DORead.enable = 0;
					DataObjOperate.Step = C_STEP_LOAD + 50;
				}
				break;

			case C_STEP_LOAD + 50:  // buffer -> main(reverse data sequence)

				for(idx=0;idx<S$LOG_MAX_SCREEN;idx++)
					{
					if(0 == idxScreen)
					{
						if(idxLog < 20)
						{
							buffer_idx = idxLog - idx - 1 ;
						}
						else
						{
							buffer_idx = S$LOG_MAX_SCREEN - idx - 1 ;
						}
					}
					else
					{
						if((idxLog-idxScreen) < 20)
						{
							buffer_idx = (idxLog-idxScreen) - idx - 1 ;
						}
						else
						{
							buffer_idx = S$LOG_MAX_SCREEN - idx - 1 ;
						}

					}
					if(buffer_idx < 0) break;
					VarLogList[buffer_idx] = VarLogList_Buffer[idx];
				}

				DataObjOperate.Step = C_STEP_LOAD + 100;

				break;

			case C_STEP_LOAD + 100:
				if(gPanelObj.vcHandle != 0)
				{
					if (!VA_Saccess(1,gPanelObj.vcHandle))
					{
						for(idx=0;idx<S$LOG_MAX_SCREEN;idx++)
							{
							pcTextlength = 30;
							if(VarLogList[idx].idxGroup == 0 && VarLogList[idx].idxText == 0)break;
							status=VA_wcGetTextByTextGroup(1,gPanelObj.vcHandle,VarLogList[idx].idxGroup,
								VarLogList[idx].idxText,(UDINT)VarNameList[idx].sText,(UDINT)&pcTextlength);
						}
						VA_Srelease(1,gPanelObj.vcHandle);
					}
				}
				DataObjOperate.Step = C_STEP_WAIT;
				break;
		}/* switch (DataObjOperate.Step) */

	}/* if(DOInfo.ident == 0 || DataObjOperate.InitStep != 3000) */

}/* end of _CYCLIC */

void fun_pv_name ()
{
	DOInfo.enable	= 1;
	DOInfo.pName 	= (UDINT)pv_get.modname;
	DatObjInfo(&DOInfo);

	if (DOInfo.status!= 0)
	{
		pv_get.errorNum = 60001; /*can not find the config data*/
		return;
	}

	if(DOInfo.len/S$LINE_LENGTH > C_PV_MAX_NO)
		{
		pv_get.errorNum = 60011; /*can not find the config data*/
		return;
	}

	while (iLine < DOInfo.len/S$LINE_LENGTH)
		{
		memcpy(&VarInfoList[iLine].pvName,(UDINT*)(DOInfo.pDatObjMem+iLine*S$LINE_LENGTH),S$LINE_LENGTH);

			status = PV_xgetadr(VarInfoList[iLine].pvName, &VarInfoList[iLine].address, &VarInfoList[iLine].length);
		if (status == 0)
		{
		}
		else if (status == 14700) /*Invalid PV name*/
		{
			break;
		}
		else if (status != 0)
		{
			pv_get.errorNum = 60111;
			pv_get.line_no  = iLine + 1;
			return;
		}

		status = PV_ninfo(VarInfoList[iLine].pvName, &VarInfoList[iLine].typ, &Length,&Dimension);
		if (status == 0)
		{
		}
		else if (status == 14700) /*Invalid PV name*/
		{
			break;
		}
		else if (status != 0)
		{
			pv_get.errorNum = 61111;
			pv_get.line_no  = iLine + 1;
			return;
		}
		iLine++;
	}/* while (iLine < DOInfo.len/S$LINE_LENGTH) */

}/* end of function */
```

#### pvgchg.typ - Local data types
```iecst
(********************************************************************
 * COPYRIGHT --  B&R China
 ********************************************************************
 * Program: pvgchg
 * File: pvgchg.typ
 * Author: lij
 * Created: March 06, 2013
 ********************************************************************
 * Local data types of program pvgchg -- point variable change log
 ********************************************************************)

TYPE
	Var_Info_typ : 	STRUCT
		pvName : STRING[C_PV_NAME_LENGTH];
		idxGroup : UINT;
		idxText : UINT;
		address : UDINT;
		length : UDINT;
		typ : UDINT;
		pValue : ARRAY[0..3]OF SINT;
	END_STRUCT;
	Var_Log_typ : 	STRUCT
		idxGroup : UINT;
		idxText : UINT;
		oldValue : STRING[11];
		curValue : STRING[11];
		chgTime : STRING[19];
	END_STRUCT;
	Var_Name_typ : 	STRUCT
		sText : ARRAY[0..29]OF UINT;
	END_STRUCT;
END_TYPE
```

#### pvchg.var
```iecst
(*array length constant*)
VAR CONSTANT
	C_PV_NAME_LENGTH : USINT := 45;
	C_PV_MAX_NO : UINT := 599;
	C_MAX_LOG__SCREEN : UINT := 19;
END_VAR
(*Task variables*)
VAR
	pv_get : pv_get_typ;
	iLine : UINT;
	VarInfoList : ARRAY[0..C_PV_MAX_NO] OF Var_Info_typ;
	status : UINT;
	Dimension : UINT;
	Length : UDINT;
	DataObjOperate : DatObj_Operate_typ;
	DOCreate : DatObjCreate;
	DOWrite : DatObjWrite;
	DORead : DatObjRead;
	DOInfo : DatObjInfo;
	VarLog : Var_Log_typ;
	pvChange : BOOL;
	idxLog : UDINT;
	VarLogList : ARRAY[0..C_MAX_LOG__SCREEN] OF Var_Log_typ;
	VarNameList : ARRAY[0..C_MAX_LOG__SCREEN] OF Var_Name_typ;
	VarLogList_Buffer : ARRAY[0..C_MAX_LOG__SCREEN] OF Var_Log_typ;
	VarNameList_Buffer : ARRAY[0..C_MAX_LOG__SCREEN] OF Var_Name_typ;
	pcTextlength : UDINT;
	idxScreen : UDINT;
	CmdPageUp : BOOL;
	CmdPageDown : BOOL;
	oldIdxLog : UDINT;
	status_tmpalloc : UINT;
	status_tmpfree : UINT;
	CmdDelete : BOOL;
	bRefresh : BOOL;
	pData : REFERENCE TO UDINT;
	OldF7 : USINT;
	OldF6 : USINT;
END_VAR
```

- edge.h (reference to Logical/GlobalIncludes/edge.h)

### Data object Logical/VarChgLog/pv_chg (Simple, version 1.00.0) - variable monitor configuration

#### pv_chg.dat
```
;********************************************************************************************
;var,array or struct configuration!
;********************************************************************************************
;fill the blank up to 45 chars and cann't use'tab' key
;maxmim 600 lines
;								                 index of text group
;								                  |
;								                  |   index of text in text group
;"                                             "  |    |
;*********** pv name ************                 |    |
"gMachinePara.MoldL.Carriage.V_Bw             ",0011,0000,;01
"gMachinePara.MoldL.Carriage.V_BwSlow         ",0011,0001,;02
"gMachinePara.MoldL.Carriage.V_BwHold         ",0011,0002,;03
"gMachinePara.MoldL.Carriage.P_Bw             ",0011,0003,;04
"gMachinePara.MoldL.Carriage.P_BwSlow         ",0011,0004,;05
"gMachinePara.MoldL.Carriage.P_BwHold         ",0011,0005,;06
"gMachinePara.MoldL.Carriage.S_Bw             ",0011,0006,;07
"gMachinePara.MoldL.Carriage.S_BwCreep        ",0011,0007,;08
"gMachinePara.MoldL.Carriage.V_Fw             ",0011,0008,;09
"gMachinePara.MoldL.Carriage.V_FwSlow         ",0011,0009,;10
"gMachinePara.MoldL.Carriage.V_FwHold         ",0011,0010,;11
"gMachinePara.MoldL.Carriage.P_Fw             ",0011,0011,;12
"gMachinePara.MoldL.Carriage.P_FwSlow         ",0011,0012,;13
"gMachinePara.MoldL.Carriage.P_FwHold         ",0011,0013,;14
"gMachinePara.MoldL.Carriage.S_Fw             ",0011,0014,;15
"gMachinePara.MoldL.Carriage.S_FwCreep        ",0011,0015,;16
"gMachinePara.MoldR.Carriage.V_Bw             ",0011,0016,;17
"gMachinePara.MoldR.Carriage.V_BwSlow         ",0011,0017,;18
"gMachinePara.MoldR.Carriage.V_BwHold         ",0011,0018,;19
"gMachinePara.MoldR.Carriage.P_Bw             ",0011,0019,;20
"gMachinePara.MoldR.Carriage.P_BwSlow         ",0011,0020,;21
"gMachinePara.MoldR.Carriage.P_BwHold         ",0011,0021,;22
"gMachinePara.MoldR.Carriage.S_Bw             ",0011,0022,;23
"gMachinePara.MoldR.Carriage.S_BwCreep        ",0011,0023,;24
"gMachinePara.MoldR.Carriage.V_Fw             ",0011,0024,;25
"gMachinePara.MoldR.Carriage.V_FwSlow         ",0011,0025,;26
"gMachinePara.MoldR.Carriage.V_FwHold         ",0011,0026,;27
"gMachinePara.MoldR.Carriage.P_Fw             ",0011,0027,;28
"gMachinePara.MoldR.Carriage.P_FwSlow         ",0011,0028,;29
"gMachinePara.MoldR.Carriage.P_FwHold         ",0011,0029,;30
"gMachinePara.MoldR.Carriage.S_Fw             ",0011,0030,;31
"gMachinePara.MoldR.Carriage.S_FwCreep        ",0011,0031,;32
"gMachinePara.MoldL.Clamp.V_Opn               ",0011,0032,;33
"gMachinePara.MoldL.Clamp.V_OpnSlow           ",0011,0033,;34
"gMachinePara.MoldL.Clamp.P_Opn               ",0011,0034,;35
"gMachinePara.MoldL.Clamp.P_OpnSlow           ",0011,0035,;36
"gMachinePara.MoldL.Clamp.S_SubMoldOut        ",0011,0036,;37
"gMachinePara.MoldL.Clamp.S_SubMoldIn         ",0011,0037,;38
"gMachinePara.MoldL.Clamp.S_OpnSlow           ",0011,0038,;39
"gMachinePara.MoldL.Clamp.S_OpnEnd            ",0011,0039,;40
"gMachinePara.MoldL.Clamp.V_Cls               ",0011,0040,;41
"gMachinePara.MoldL.Clamp.V_ClsSlow           ",0011,0041,;42
"gMachinePara.MoldL.Clamp.V_Tonnage           ",0011,0042,;43
"gMachinePara.MoldL.Clamp.P_Cls               ",0011,0043,;44
"gMachinePara.MoldL.Clamp.P_ClsSlow           ",0011,0044,;45
"gMachinePara.MoldL.Clamp.P_Tonnage           ",0011,0045,;46
"gMachinePara.MoldL.Clamp.S_Cls               ",0011,0046,;47
"gMachinePara.MoldL.Clamp.S_ClsEnd            ",0011,0047,;48
"gMachinePara.MoldR.Clamp.V_Opn               ",0011,0048,;49
"gMachinePara.MoldR.Clamp.V_OpnSlow           ",0011,0049,;50
"gMachinePara.MoldR.Clamp.P_Opn               ",0011,0050,;51
"gMachinePara.MoldR.Clamp.P_OpnSlow           ",0011,0051,;52
"gMachinePara.MoldR.Clamp.S_SubMoldOut        ",0011,0052,;53
"gMachinePara.MoldR.Clamp.S_SubMoldIn         ",0011,0053,;54
"gMachinePara.MoldR.Clamp.S_OpnSlow           ",0011,0054,;55
"gMachinePara.MoldR.Clamp.S_OpnEnd            ",0011,0055,;56
"gMachinePara.MoldR.Clamp.V_Cls               ",0011,0056,;57
"gMachinePara.MoldR.Clamp.V_ClsSlow           ",0011,0057,;58
"gMachinePara.MoldR.Clamp.V_Tonnage           ",0011,0058,;59
"gMachinePara.MoldR.Clamp.P_Cls               ",0011,0059,;60
"gMachinePara.MoldR.Clamp.P_ClsSlow           ",0011,0060,;61
"gMachinePara.MoldR.Clamp.P_Tonnage           ",0011,0061,;62
"gMachinePara.MoldR.Clamp.S_Cls               ",0011,0062,;63
"gMachinePara.MoldR.Clamp.S_ClsEnd            ",0011,0063,;64
"gMachinePara.MoldL.BlowPin.V_Up              ",0011,0064,;65
"gMachinePara.MoldL.BlowPin.V_UpMicro         ",0011,0065,;66
"gMachinePara.MoldL.BlowPin.P_Up              ",0011,0066,;67
"gMachinePara.MoldL.BlowPin.P_UpMicro         ",0011,0067,;68
"gMachinePara.MoldL.BlowPin.S_Up              ",0011,0068,;69
"gMachinePara.MoldL.BlowPin.S_UpMicro         ",0011,0069,;70
"gMachinePara.MoldL.BlowPin.V_Dn              ",0011,0070,;71
"gMachinePara.MoldL.BlowPin.V_DnSlow          ",0011,0071,;72
"gMachinePara.MoldL.BlowPin.P_Dn              ",0011,0072,;73
"gMachinePara.MoldL.BlowPin.P_DnSlow          ",0011,0073,;74
"gMachinePara.MoldL.BlowPin.S_Dn              ",0011,0074,;75
"gMachinePara.MoldL.BlowPin.S_DnSlow          ",0011,0075,;76
"gMachinePara.MoldR.BlowPin.V_Up              ",0011,0076,;77
"gMachinePara.MoldR.BlowPin.V_UpMicro         ",0011,0077,;78
"gMachinePara.MoldR.BlowPin.P_Up              ",0011,0078,;79
"gMachinePara.MoldR.BlowPin.P_UpMicro         ",0011,0079,;80
"gMachinePara.MoldR.BlowPin.S_Up              ",0011,0080,;81
"gMachinePara.MoldR.BlowPin.S_UpMicro         ",0011,0081,;82
"gMachinePara.MoldR.BlowPin.V_Dn              ",0011,0082,;83
"gMachinePara.MoldR.BlowPin.V_DnSlow          ",0011,0083,;84
"gMachinePara.MoldR.BlowPin.P_Dn              ",0011,0084,;85
"gMachinePara.MoldR.BlowPin.P_DnSlow          ",0011,0085,;86
"gMachinePara.MoldR.BlowPin.S_Dn              ",0011,0086,;87
"gMachinePara.MoldR.BlowPin.S_DnSlow          ",0011,0087,;88
"gMachineFix.MoldL.Carriage.Fw.accel          ",0011,0088,;89
"gMachineFix.MoldL.Carriage.Fw.decel          ",0011,0089,;90
"gMachineFix.MoldL.Carriage.Fw.decel_end      ",0011,0090,;91
"gMachineFix.MoldL.Carriage.Fw.Tj             ",0011,0091,;92
"gMachineFix.MoldL.Carriage.Fw.Td             ",0011,0092,;93
"gMachineFix.MoldR.Carriage.Fw.accel          ",0011,0093,;94
"gMachineFix.MoldR.Carriage.Fw.decel          ",0011,0094,;95
"gMachineFix.MoldR.Carriage.Fw.decel_end      ",0011,0095,;96
"gMachineFix.MoldR.Carriage.Fw.Tj             ",0011,0096,;97
"gMachineFix.MoldR.Carriage.Fw.Td             ",0011,0097,;98
"gMachineFix.MoldL.Carriage.Bw.accel          ",0011,0098,;99
"gMachineFix.MoldL.Carriage.Bw.decel          ",0011,0099,;100
"gMachineFix.MoldL.Carriage.Bw.decel_end      ",0011,0100,;101
"gMachineFix.MoldL.Carriage.Bw.Tj             ",0011,0101,;102
"gMachineFix.MoldL.Carriage.Bw.Td             ",0011,0102,;103
"gMachineFix.MoldR.Carriage.Bw.accel          ",0011,0103,;104
"gMachineFix.MoldR.Carriage.Bw.decel          ",0011,0104,;105
"gMachineFix.MoldR.Carriage.Bw.decel_end      ",0011,0105,;106
"gMachineFix.MoldR.Carriage.Bw.Tj             ",0011,0106,;107
"gMachineFix.MoldR.Carriage.Bw.Td             ",0011,0107,;108
"gMachineFix.MoldL.Clamp.Close.accel          ",0011,0108,;109
"gMachineFix.MoldL.Clamp.Close.decel          ",0011,0109,;110
"gMachineFix.MoldL.Clamp.Close.decel_end      ",0011,0110,;111
"gMachineFix.MoldL.Clamp.Close.Tj             ",0011,0111,;112
"gMachineFix.MoldL.Clamp.Close.Td             ",0011,0112,;113
"gMachineFix.MoldR.Clamp.Close.accel          ",0011,0113,;114
"gMachineFix.MoldR.Clamp.Close.decel          ",0011,0114,;115
"gMachineFix.MoldR.Clamp.Close.decel_end      ",0011,0115,;116
"gMachineFix.MoldR.Clamp.Close.Tj             ",0011,0116,;117
"gMachineFix.MoldR.Clamp.Close.Td             ",0011,0117,;118
"gMachineFix.MoldL.Clamp.Open.accel           ",0011,0118,;119
"gMachineFix.MoldL.Clamp.Open.decel           ",0011,0119,;120
"gMachineFix.MoldL.Clamp.Open.decel_end       ",0011,0120,;121
"gMachineFix.MoldL.Clamp.Open.Tj              ",0011,0121,;122
"gMachineFix.MoldL.Clamp.Open.Td              ",0011,0122,;123
"gMachineFix.MoldR.Clamp.Open.accel           ",0011,0123,;124
"gMachineFix.MoldR.Clamp.Open.decel           ",0011,0124,;125
"gMachineFix.MoldR.Clamp.Open.decel_end       ",0011,0125,;126
"gMachineFix.MoldR.Clamp.Open.Tj              ",0011,0126,;127
"gMachineFix.MoldR.Clamp.Open.Td              ",0011,0127,;128
"gMachineFix.MoldL.BlowPin.Down.accel         ",0011,0128,;129
"gMachineFix.MoldL.BlowPin.Down.decel         ",0011,0129,;130
"gMachineFix.MoldL.BlowPin.Down.decel_end     ",0011,0130,;131
"gMachineFix.MoldL.BlowPin.Down.Tj            ",0011,0131,;132
"gMachineFix.MoldL.BlowPin.Down.Td            ",0011,0132,;133
"gMachineFix.MoldR.BlowPin.Down.accel         ",0011,0133,;134
"gMachineFix.MoldR.BlowPin.Down.decel         ",0011,0134,;135
"gMachineFix.MoldR.BlowPin.Down.decel_end     ",0011,0135,;136
"gMachineFix.MoldR.BlowPin.Down.Tj            ",0011,0136,;137
"gMachineFix.MoldR.BlowPin.Down.Td            ",0011,0137,;138
"gMachineFix.MoldL.BlowPin.Up.accel           ",0011,0138,;139
"gMachineFix.MoldL.BlowPin.Up.decel           ",0011,0139,;140
"gMachineFix.MoldL.BlowPin.Up.decel_end       ",0011,0140,;141
"gMachineFix.MoldL.BlowPin.Up.Tj              ",0011,0141,;142
"gMachineFix.MoldL.BlowPin.Up.Td              ",0011,0142,;143
"gMachineFix.MoldR.BlowPin.Up.accel           ",0011,0143,;144
"gMachineFix.MoldR.BlowPin.Up.decel           ",0011,0144,;145
"gMachineFix.MoldR.BlowPin.Up.decel_end       ",0011,0145,;146
"gMachineFix.MoldR.BlowPin.Up.Tj              ",0011,0146,;147
"gMachineFix.MoldR.BlowPin.Up.Td              ",0011,0147,;148
"gMachineFix.MoldL.Clamp.Close.VoltageMin     ",0011,0148,;149
"gMachineFix.MoldL.Clamp.Close.VoltageMax     ",0011,0149,;150
"gMachineFix.MoldL.Clamp.Close.V_Max          ",0011,0150,;151
"gMachineFix.MoldL.Clamp.Open.VoltageMin      ",0011,0151,;152
"gMachineFix.MoldL.Clamp.Open.VoltageMax      ",0011,0152,;153
"gMachineFix.MoldL.Clamp.Open.V_Max           ",0011,0153,;154
"gMachineFix.MoldR.Clamp.Close.VoltageMin     ",0011,0154,;155
"gMachineFix.MoldR.Clamp.Close.VoltageMax     ",0011,0155,;156
"gMachineFix.MoldR.Clamp.Close.V_Max          ",0011,0156,;157
"gMachineFix.MoldR.Clamp.Open.VoltageMin      ",0011,0157,;158
"gMachineFix.MoldR.Clamp.Open.VoltageMax      ",0011,0158,;159
"gMachineFix.MoldR.Clamp.Open.V_Max           ",0011,0159,;160
"gMachineFix.MoldL.Carriage.Fw.VoltageMin     ",0011,0160,;161
"gMachineFix.MoldL.Carriage.Fw.VoltageMax     ",0011,0161,;162
"gMachineFix.MoldL.Carriage.Fw.V_Max          ",0011,0162,;163
"gMachineFix.MoldL.Carriage.Bw.VoltageMin     ",0011,0163,;164
"gMachineFix.MoldL.Carriage.Bw.VoltageMax     ",0011,0164,;165
"gMachineFix.MoldL.Carriage.Bw.V_Max          ",0011,0165,;166
"gMachineFix.MoldR.Carriage.Fw.VoltageMin     ",0011,0166,;167
"gMachineFix.MoldR.Carriage.Fw.VoltageMax     ",0011,0167,;168
"gMachineFix.MoldR.Carriage.Fw.V_Max          ",0011,0168,;169
"gMachineFix.MoldR.Carriage.Bw.VoltageMin     ",0011,0169,;170
"gMachineFix.MoldR.Carriage.Bw.VoltageMax     ",0011,0170,;171
"gMachineFix.MoldR.Carriage.Bw.V_Max          ",0011,0171,;172
"gMachineFix.MoldL.Clamp.Zero                 ",0011,0172,;173
"gMachineFix.MoldL.Clamp.Max                  ",0011,0173,;174
"gMachineFix.MoldL.Clamp.Length               ",0011,0174,;175
"gMachineFix.MoldR.Clamp.Zero                 ",0011,0175,;176
"gMachineFix.MoldR.Clamp.Max                  ",0011,0176,;177
"gMachineFix.MoldR.Clamp.Length               ",0011,0177,;178
"gMachineFix.MoldL.Carriage.Zero              ",0011,0178,;179
"gMachineFix.MoldL.Carriage.Max               ",0011,0179,;180
"gMachineFix.MoldL.Carriage.Length            ",0011,0180,;181
"gMachineFix.MoldR.Carriage.Zero              ",0011,0181,;182
"gMachineFix.MoldR.Carriage.Max               ",0011,0182,;183
"gMachineFix.MoldR.Carriage.Length            ",0011,0183,;184
"gMachineFix.MoldR.Clamp.Tolerance            ",0011,0184,;185
"gMachineFix.MoldR.Carriage.Tolerance         ",0011,0185,;186
```

### Package Logical/Motion - Axis part

### Data object Logical/Motion/acp10etxen (Ett)

- acp10etxen.ett (not shown)

### Data object Logical/Motion/init/UpDnR (Ax)

#### UpDnR.ax
```
InitParameter (Version=2.48.1, NcSwId=ACP10)
  ACP10AXIS_typ:
    dig_in:
      level:
        reference = ncACTIV_HI
        pos_hw_end = ncACTIV_HI
        neg_hw_end = ncACTIV_HI
        trigger1 = ncACTIV_HI
        trigger2 = ncACTIV_HI + ncQUICKSTOP
    encoder_if:
      parameter:
        count_dir = ncSTANDARD
        scaling:
          load:
            units = 1600
            rev_motor = 1
    limit:
      parameter:
        v_pos = 96000.0
        v_neg = 96000.0
        a1_pos = 960000.0
        a2_pos = 960000.0
        a1_neg = 960000.0
        a2_neg = 960000.0
        t_jolt = 0.1
        t_in_pos = 0.0
        pos_sw_end = 8388607
        neg_sw_end = -8388608
        ds_warning = 800.0
        ds_stop = 16000.0
        a_stop = 1.0e+30
        dv_stop = 0.0
        dv_stop_mode = ncOFF
    controller:
      mode = ncPOSITION
      position:
        kv = 540.0
        tn = 0.0
        t_predict = 0.0004
        t_total = 0.0004
        p_max = 1.0e+30
        i_max = 0.0
      speed:
        kv = 1.2
        tn = 0.0
        t_filter = 0.0
        isq_filter1:
          type = ncOFF
          a0 = 0.0
          a1 = 0.0
          b0 = 0.0
          b1 = 0.0
          b2 = 0.0
          c0_par_id = 0
          c1_par_id = 0
        isq_filter2:
          type = ncOFF
          a0 = 0.0
          a1 = 0.0
          b0 = 0.0
          b1 = 0.0
          b2 = 0.0
          c0_par_id = 0
          c1_par_id = 0
        isq_filter3:
          type = ncOFF
          a0 = 0.0
          a1 = 0.0
          b0 = 0.0
          b1 = 0.0
          b2 = 0.0
          c0_par_id = 0
          c1_par_id = 0
      uf:
        type = ncLINEAR
        auto_config = ncMOTOR_PAR
        u0 = 0.0
        un = 0.0
        fn = 50.0
        k_f_slip = 0.0
      ff:
        torque_load = 0.0
        torque_pos = 0.0
        torque_neg = 0.0
        kv_torque = 0.0
        inertia = 0.0
        t_filter_a = 0.0
    move:
      stop:
        parameter[0]:
          decel_ramp = ncA_LIMIT
          controller = ncON
        parameter[1]:
          decel_ramp = ncA_LIMIT
          controller = ncON
        parameter[2]:
          decel_ramp = ncA_LIMIT
          controller = ncON
        parameter[3]:
          decel_ramp = ncA_LIMIT
          controller = ncON
        quickstop:
          decel_ramp = ncA_LIMIT
        drive_error:
          decel_ramp = ncA_LIMIT
      homing:
        parameter:
          s = 0
          v_switch = 5000.0
          v_trigger = 500.0
          a = 50000.0
          mode = ncDIRECT
          edge_sw = ncPOSITIVE
          start_dir = ncPOSITIVE
          trigg_dir = ncPOSITIVE
          ref_pulse = ncOFF
          fix_dir = ncOFF
          tr_s_block = 0.0
          torque_lim = 0.0
          ds_block = 0.0
          ds_stop = 0.0
      basis:
        parameter:
          v_pos = 5000.0
          v_neg = 5000.0
          a1_pos = 50000.0
          a2_pos = 50000.0
          a1_neg = 50000.0
          a2_neg = 50000.0
    message:
      text:
        parameter:
          format = ncBREAK
          columns = 80
          data_modul = acp10etxen
```

### Data object Logical/Motion/init/UpDnL (Ax)

#### UpDnL.ax
```
InitParameter (Version=2.48.1, NcSwId=ACP10)
  ACP10AXIS_typ:
    dig_in:
      level:
        reference = ncACTIV_HI
        pos_hw_end = ncACTIV_HI
        neg_hw_end = ncACTIV_HI
        trigger1 = ncACTIV_HI
        trigger2 = ncACTIV_HI + ncQUICKSTOP
    encoder_if:
      parameter:
        count_dir = ncSTANDARD
        scaling:
          load:
            units = 1600
            rev_motor = 1
    limit:
      parameter:
        v_pos = 96000.0
        v_neg = 96000.0
        a1_pos = 960000.0
        a2_pos = 960000.0
        a1_neg = 960000.0
        a2_neg = 960000.0
        t_jolt = 0.1
        t_in_pos = 0.0
        pos_sw_end = 8388607
        neg_sw_end = -8388608
        ds_warning = 800.0
        ds_stop = 1600.0
        a_stop = 1.0E+30
        dv_stop = 0.0
        dv_stop_mode = ncOFF
    controller:
      mode = ncPOSITION
      position:
        kv = 520.0
        tn = 0.0
        t_predict = 0.0004
        t_total = 0.0004
        p_max = 1.0E+30
        i_max = 0.0
      speed:
        kv = 0.85
        tn = 0.0
        t_filter = 0.0
        isq_filter1:
          type = ncOFF
          a0 = 0.0
          a1 = 0.0
          b0 = 0.0
          b1 = 0.0
          b2 = 0.0
          c0_par_id = 0
          c1_par_id = 0
        isq_filter2:
          type = ncOFF
          a0 = 0.0
          a1 = 0.0
          b0 = 0.0
          b1 = 0.0
          b2 = 0.0
          c0_par_id = 0
          c1_par_id = 0
        isq_filter3:
          type = ncOFF
          a0 = 0.0
          a1 = 0.0
          b0 = 0.0
          b1 = 0.0
          b2 = 0.0
          c0_par_id = 0
          c1_par_id = 0
      uf:
        type = ncLINEAR
        auto_config = ncMOTOR_PAR
        u0 = 0.0
        un = 0.0
        fn = 50.0
        k_f_slip = 0.0
      ff:
        torque_load = 0.0
        torque_pos = 0.0
        torque_neg = 0.0
        kv_torque = 0.0
        inertia = 0.0
        t_filter_a = 0.0
    move:
      stop:
        parameter[0]:
          decel_ramp = ncA_LIMIT
          controller = ncON
        parameter[1]:
          decel_ramp = ncA_LIMIT
          controller = ncON
        parameter[2]:
          decel_ramp = ncA_LIMIT
          controller = ncON
        parameter[3]:
          decel_ramp = ncA_LIMIT
          controller = ncON
        quickstop:
          decel_ramp = ncA_LIMIT
        drive_error:
          decel_ramp = ncA_LIMIT
      homing:
        parameter:
          s = 0
          v_switch = 5000.0
          v_trigger = 500.0
          a = 50000.0
          mode = ncDIRECT
          edge_sw = ncPOSITIVE
          start_dir = ncPOSITIVE
          trigg_dir = ncPOSITIVE
          ref_pulse = ncOFF
          fix_dir = ncOFF
          tr_s_block = 0.0
          torque_lim = 0.0
          ds_block = 0.0
          ds_stop = 0.0
      basis:
        parameter:
          v_pos = 5000.0
          v_neg = 5000.0
          a1_pos = 50000.0
          a2_pos = 50000.0
          a1_neg = 50000.0
          a2_neg = 50000.0
    message:
      text:
        parameter:
          format = ncBREAK
          columns = 80
          data_modul = acp10etxen
```

### Data object Logical/Motion/init/TransferR (Ax)

#### TransferR.ax
```
InitParameter (Version=5.06.1, NcSwId=ACP10)
  ACP10AXIS_typ:
    dig_in:
      level:
        reference = ncACTIV_HI
        pos_hw_end = ncACTIV_HI
        neg_hw_end = ncACTIV_HI
        trigger1 = ncACTIV_HI
        trigger2 = ncACTIV_HI + ncQUICKSTOP
    encoder_if:
      parameter:
        count_dir = ncSTANDARD
        scaling:
          load:
            units = 2500
            rev_motor = 1
    limit:
      parameter:
        v_pos = 125000.0
        v_neg = 125000.0
        a1_pos = 500000.0
        a2_pos = 500000.0
        a1_neg = 500000.0
        a2_neg = 500000.0
        t_jolt = 0.1
        t_in_pos = 0.0
        pos_sw_end = 8388607
        neg_sw_end = -8388608
        ds_warning = 625.0
        ds_stop = 1250.0
        a_stop = 1.0E+30
        dv_stop = 0.0
        dv_stop_mode = ncOFF
    controller:
      mode = ncPOSITION
      position:
        kv = 400.0
        tn = 0.0
        t_predict = 0.0004
        t_total = 0.0004
        p_max = 1.0E+30
        i_max = 0.0
      speed:
        kv = 1.05
        tn = 0.0
        t_filter = 0.0012
        isq_filter1:
          type = ncOFF
          a0 = 0.0
          a1 = 0.0
          b0 = 0.0
          b1 = 0.0
          b2 = 0.0
          c0_par_id = 0
          c1_par_id = 0
        isq_filter2:
          type = ncOFF
          a0 = 0.0
          a1 = 0.0
          b0 = 0.0
          b1 = 0.0
          b2 = 0.0
          c0_par_id = 0
          c1_par_id = 0
        isq_filter3:
          type = ncOFF
          a0 = 0.0
          a1 = 0.0
          b0 = 0.0
          b1 = 0.0
          b2 = 0.0
          c0_par_id = 0
          c1_par_id = 0
      uf:
        type = ncLINEAR
        auto_config = ncMOTOR_PAR
        u0 = 0.0
        un = 0.0
        fn = 50.0
        k_f_slip = 0.0
      ff:
        mode = ncSTANDARD
        torque_load = 0.0
        torque_pos = 0.0
        torque_neg = 0.0
        kv_torque = 0.0
        inertia = 0.0
        t_filter_a = 0.0
      fb:
        mode = ncSTANDARD
        speed_mix_ratio = 0.0
        speed_kv = 2.0
      model:
        mass1:
          inertia = 0
          viscous_friction = 0
        mass2:
          inertia = 0
          viscous_friction = 0
          stiffness = 0
          damping = 0
    move:
      stop:
        parameter[0]:
          decel_ramp = ncA_LIMIT
          controller = ncON
        parameter[1]:
          decel_ramp = ncA_LIMIT
          controller = ncON
        parameter[2]:
          decel_ramp = ncA_LIMIT
          controller = ncON
        parameter[3]:
          decel_ramp = ncA_LIMIT
          controller = ncON
        quickstop:
          decel_ramp = ncA_LIMIT
          t_jolt = 0
        drive_error:
          decel_ramp = ncA_LIMIT
      homing:
        parameter:
          s = 0
          v_switch = 5000.0
          v_trigger = 500.0
          a = 50000.0
          mode = ncDIRECT
          edge_sw = ncPOSITIVE
          start_dir = ncPOSITIVE
          trigg_dir = ncPOSITIVE
          ref_pulse = ncOFF
          fix_dir = ncOFF
          tr_s_block = 0.0
          torque_lim = 0.0
          ds_block = 0.0
          ds_stop = 0.0
      basis:
        parameter:
          v_pos = 5000.0
          v_neg = 5000.0
          a1_pos = 50000.0
          a2_pos = 50000.0
          a1_neg = 50000.0
          a2_neg = 50000.0
    message:
      text:
        parameter:
          format = ncBREAK
          columns = 80
          data_modul = acp10etxen
```

### Data object Logical/Motion/init/TransferL (Ax)

#### TransferL.ax
```
InitParameter (Version=5.06.1, NcSwId=ACP10)
  ACP10AXIS_typ:
    dig_in:
      level:
        reference = ncACTIV_HI
        pos_hw_end = ncACTIV_HI
        neg_hw_end = ncACTIV_HI
        trigger1 = ncACTIV_HI
        trigger2 = ncACTIV_HI + ncQUICKSTOP
    encoder_if:
      parameter:
        count_dir = ncSTANDARD
        scaling:
          load:
            units = 2500
            rev_motor = 1
    limit:
      parameter:
        v_pos = 125000.0
        v_neg = 125000.0
        a1_pos = 1500000.0
        a2_pos = 1500000.0
        a1_neg = 1500000.0
        a2_neg = 1500000.0
        t_jolt = 0.1
        t_in_pos = 0.0
        pos_sw_end = 8388607
        neg_sw_end = -8388608
        ds_warning = 625.0
        ds_stop = 1250.0
        a_stop = 1.0E+30
        dv_stop = 0.0
        dv_stop_mode = ncOFF
    controller:
      mode = ncPOSITION
      position:
        kv = 600.0
        tn = 0.0
        t_predict = 0.0004
        t_total = 0.0004
        p_max = 1.0E+30
        i_max = 0.0
      speed:
        kv = 0.9
        tn = 0.0
        t_filter = 0.0
        isq_filter1:
          type = ncOFF
          a0 = 0.0
          a1 = 0.0
          b0 = 0.0
          b1 = 0.0
          b2 = 0.0
          c0_par_id = 0
          c1_par_id = 0
        isq_filter2:
          type = ncOFF
          a0 = 0.0
          a1 = 0.0
          b0 = 0.0
          b1 = 0.0
          b2 = 0.0
          c0_par_id = 0
          c1_par_id = 0
        isq_filter3:
          type = ncOFF
          a0 = 0.0
          a1 = 0.0
          b0 = 0.0
          b1 = 0.0
          b2 = 0.0
          c0_par_id = 0
          c1_par_id = 0
      uf:
        type = ncLINEAR
        auto_config = ncMOTOR_PAR
        u0 = 0.0
        un = 0.0
        fn = 50.0
        k_f_slip = 0.0
      ff:
        mode = ncSTANDARD
        torque_load = 0.0
        torque_pos = 0.0
        torque_neg = 0.0
        kv_torque = 0.0
        inertia = 0.0
        t_filter_a = 0.0
      fb:
        mode = ncSTANDARD
        speed_mix_ratio = 0.0
        speed_kv = 2.0
      model:
        mass1:
          inertia = 0
          viscous_friction = 0
        mass2:
          inertia = 0
          viscous_friction = 0
          stiffness = 0
          damping = 0
    move:
      stop:
        parameter[0]:
          decel_ramp = ncA_LIMIT
          controller = ncON
        parameter[1]:
          decel_ramp = ncA_LIMIT
          controller = ncON
        parameter[2]:
          decel_ramp = ncA_LIMIT
          controller = ncON
        parameter[3]:
          decel_ramp = ncA_LIMIT
          controller = ncON
        quickstop:
          decel_ramp = ncA_LIMIT
          t_jolt = 0
        drive_error:
          decel_ramp = ncA_LIMIT
      homing:
        parameter:
          s = 0
          v_switch = 5000.0
          v_trigger = 500.0
          a = 50000.0
          mode = ncDIRECT
          edge_sw = ncPOSITIVE
          start_dir = ncPOSITIVE
          trigg_dir = ncPOSITIVE
          ref_pulse = ncOFF
          fix_dir = ncOFF
          tr_s_block = 0.0
          torque_lim = 0.0
          ds_block = 0.0
          ds_stop = 0.0
      basis:
        parameter:
          v_pos = 5000.0
          v_neg = 5000.0
          a1_pos = 50000.0
          a2_pos = 50000.0
          a1_neg = 50000.0
          a2_neg = 50000.0
    message:
      text:
        parameter:
          format = ncBREAK
          columns = 80
          data_modul = acp10etxen
```

### Data object Logical/Motion/init/ClampR (Ax)
